(* IEC 61131-3 sources: AXOpen/src/showcase/app/SystemConstants (part 4) *)

TYPE
    kuka_rb1_DIO512_Output_Layout : STRUCT
        Signals_64_0 AT %X0.0 : BOOL;
        Signals_64_1 AT %X0.1 : BOOL;
        Signals_64_2 AT %X0.2 : BOOL;
        Signals_64_3 AT %X0.3 : BOOL;
        Signals_64_4 AT %X0.4 : BOOL;
        Signals_64_5 AT %X0.5 : BOOL;
        Signals_64_6 AT %X0.6 : BOOL;
        Signals_64_7 AT %X0.7 : BOOL;
        Signals_65_0 AT %X1.0 : BOOL;
        Signals_65_1 AT %X1.1 : BOOL;
        Signals_65_2 AT %X1.2 : BOOL;
        Signals_65_3 AT %X1.3 : BOOL;
        Signals_65_4 AT %X1.4 : BOOL;
        Signals_65_5 AT %X1.5 : BOOL;
        Signals_65_6 AT %X1.6 : BOOL;
        Signals_65_7 AT %X1.7 : BOOL;
        Signals_66_0 AT %X2.0 : BOOL;
        Signals_66_1 AT %X2.1 : BOOL;
        Signals_66_2 AT %X2.2 : BOOL;
        Signals_66_3 AT %X2.3 : BOOL;
        Signals_66_4 AT %X2.4 : BOOL;
        Signals_66_5 AT %X2.5 : BOOL;
        Signals_66_6 AT %X2.6 : BOOL;
        Signals_66_7 AT %X2.7 : BOOL;
        Signals_67_0 AT %X3.0 : BOOL;
        Signals_67_1 AT %X3.1 : BOOL;
        Signals_67_2 AT %X3.2 : BOOL;
        Signals_67_3 AT %X3.3 : BOOL;
        Signals_67_4 AT %X3.4 : BOOL;
        Signals_67_5 AT %X3.5 : BOOL;
        Signals_67_6 AT %X3.6 : BOOL;
        Signals_67_7 AT %X3.7 : BOOL;
        Signals_68_0 AT %X4.0 : BOOL;
        Signals_68_1 AT %X4.1 : BOOL;
        Signals_68_2 AT %X4.2 : BOOL;
        Signals_68_3 AT %X4.3 : BOOL;
        Signals_68_4 AT %X4.4 : BOOL;
        Signals_68_5 AT %X4.5 : BOOL;
        Signals_68_6 AT %X4.6 : BOOL;
        Signals_68_7 AT %X4.7 : BOOL;
        Signals_69_0 AT %X5.0 : BOOL;
        Signals_69_1 AT %X5.1 : BOOL;
        Signals_69_2 AT %X5.2 : BOOL;
        Signals_69_3 AT %X5.3 : BOOL;
        Signals_69_4 AT %X5.4 : BOOL;
        Signals_69_5 AT %X5.5 : BOOL;
        Signals_69_6 AT %X5.6 : BOOL;
        Signals_69_7 AT %X5.7 : BOOL;
        Signals_70_0 AT %X6.0 : BOOL;
        Signals_70_1 AT %X6.1 : BOOL;
        Signals_70_2 AT %X6.2 : BOOL;
        Signals_70_3 AT %X6.3 : BOOL;
        Signals_70_4 AT %X6.4 : BOOL;
        Signals_70_5 AT %X6.5 : BOOL;
        Signals_70_6 AT %X6.6 : BOOL;
        Signals_70_7 AT %X6.7 : BOOL;
        Signals_71_0 AT %X7.0 : BOOL;
        Signals_71_1 AT %X7.1 : BOOL;
        Signals_71_2 AT %X7.2 : BOOL;
        Signals_71_3 AT %X7.3 : BOOL;
        Signals_71_4 AT %X7.4 : BOOL;
        Signals_71_5 AT %X7.5 : BOOL;
        Signals_71_6 AT %X7.6 : BOOL;
        Signals_71_7 AT %X7.7 : BOOL;
        Signals_72_0 AT %X8.0 : BOOL;
        Signals_72_1 AT %X8.1 : BOOL;
        Signals_72_2 AT %X8.2 : BOOL;
        Signals_72_3 AT %X8.3 : BOOL;
        Signals_72_4 AT %X8.4 : BOOL;
        Signals_72_5 AT %X8.5 : BOOL;
        Signals_72_6 AT %X8.6 : BOOL;
        Signals_72_7 AT %X8.7 : BOOL;
        Signals_73_0 AT %X9.0 : BOOL;
        Signals_73_1 AT %X9.1 : BOOL;
        Signals_73_2 AT %X9.2 : BOOL;
        Signals_73_3 AT %X9.3 : BOOL;
        Signals_73_4 AT %X9.4 : BOOL;
        Signals_73_5 AT %X9.5 : BOOL;
        Signals_73_6 AT %X9.6 : BOOL;
        Signals_73_7 AT %X9.7 : BOOL;
        Signals_74_0 AT %X10.0 : BOOL;
        Signals_74_1 AT %X10.1 : BOOL;
        Signals_74_2 AT %X10.2 : BOOL;
        Signals_74_3 AT %X10.3 : BOOL;
        Signals_74_4 AT %X10.4 : BOOL;
        Signals_74_5 AT %X10.5 : BOOL;
        Signals_74_6 AT %X10.6 : BOOL;
        Signals_74_7 AT %X10.7 : BOOL;
        Signals_75_0 AT %X11.0 : BOOL;
        Signals_75_1 AT %X11.1 : BOOL;
        Signals_75_2 AT %X11.2 : BOOL;
        Signals_75_3 AT %X11.3 : BOOL;
        Signals_75_4 AT %X11.4 : BOOL;
        Signals_75_5 AT %X11.5 : BOOL;
        Signals_75_6 AT %X11.6 : BOOL;
        Signals_75_7 AT %X11.7 : BOOL;
        Signals_76_0 AT %X12.0 : BOOL;
        Signals_76_1 AT %X12.1 : BOOL;
        Signals_76_2 AT %X12.2 : BOOL;
        Signals_76_3 AT %X12.3 : BOOL;
        Signals_76_4 AT %X12.4 : BOOL;
        Signals_76_5 AT %X12.5 : BOOL;
        Signals_76_6 AT %X12.6 : BOOL;
        Signals_76_7 AT %X12.7 : BOOL;
        Signals_77_0 AT %X13.0 : BOOL;
        Signals_77_1 AT %X13.1 : BOOL;
        Signals_77_2 AT %X13.2 : BOOL;
        Signals_77_3 AT %X13.3 : BOOL;
        Signals_77_4 AT %X13.4 : BOOL;
        Signals_77_5 AT %X13.5 : BOOL;
        Signals_77_6 AT %X13.6 : BOOL;
        Signals_77_7 AT %X13.7 : BOOL;
        Signals_78_0 AT %X14.0 : BOOL;
        Signals_78_1 AT %X14.1 : BOOL;
        Signals_78_2 AT %X14.2 : BOOL;
        Signals_78_3 AT %X14.3 : BOOL;
        Signals_78_4 AT %X14.4 : BOOL;
        Signals_78_5 AT %X14.5 : BOOL;
        Signals_78_6 AT %X14.6 : BOOL;
        Signals_78_7 AT %X14.7 : BOOL;
        Signals_79_0 AT %X15.0 : BOOL;
        Signals_79_1 AT %X15.1 : BOOL;
        Signals_79_2 AT %X15.2 : BOOL;
        Signals_79_3 AT %X15.3 : BOOL;
        Signals_79_4 AT %X15.4 : BOOL;
        Signals_79_5 AT %X15.5 : BOOL;
        Signals_79_6 AT %X15.6 : BOOL;
        Signals_79_7 AT %X15.7 : BOOL;
        Signals_80_0 AT %X16.0 : BOOL;
        Signals_80_1 AT %X16.1 : BOOL;
        Signals_80_2 AT %X16.2 : BOOL;
        Signals_80_3 AT %X16.3 : BOOL;
        Signals_80_4 AT %X16.4 : BOOL;
        Signals_80_5 AT %X16.5 : BOOL;
        Signals_80_6 AT %X16.6 : BOOL;
        Signals_80_7 AT %X16.7 : BOOL;
        Signals_81_0 AT %X17.0 : BOOL;
        Signals_81_1 AT %X17.1 : BOOL;
        Signals_81_2 AT %X17.2 : BOOL;
        Signals_81_3 AT %X17.3 : BOOL;
        Signals_81_4 AT %X17.4 : BOOL;
        Signals_81_5 AT %X17.5 : BOOL;
        Signals_81_6 AT %X17.6 : BOOL;
        Signals_81_7 AT %X17.7 : BOOL;
        Signals_82_0 AT %X18.0 : BOOL;
        Signals_82_1 AT %X18.1 : BOOL;
        Signals_82_2 AT %X18.2 : BOOL;
        Signals_82_3 AT %X18.3 : BOOL;
        Signals_82_4 AT %X18.4 : BOOL;
        Signals_82_5 AT %X18.5 : BOOL;
        Signals_82_6 AT %X18.6 : BOOL;
        Signals_82_7 AT %X18.7 : BOOL;
        Signals_83_0 AT %X19.0 : BOOL;
        Signals_83_1 AT %X19.1 : BOOL;
        Signals_83_2 AT %X19.2 : BOOL;
        Signals_83_3 AT %X19.3 : BOOL;
        Signals_83_4 AT %X19.4 : BOOL;
        Signals_83_5 AT %X19.5 : BOOL;
        Signals_83_6 AT %X19.6 : BOOL;
        Signals_83_7 AT %X19.7 : BOOL;
        Signals_84_0 AT %X20.0 : BOOL;
        Signals_84_1 AT %X20.1 : BOOL;
        Signals_84_2 AT %X20.2 : BOOL;
        Signals_84_3 AT %X20.3 : BOOL;
        Signals_84_4 AT %X20.4 : BOOL;
        Signals_84_5 AT %X20.5 : BOOL;
        Signals_84_6 AT %X20.6 : BOOL;
        Signals_84_7 AT %X20.7 : BOOL;
        Signals_85_0 AT %X21.0 : BOOL;
        Signals_85_1 AT %X21.1 : BOOL;
        Signals_85_2 AT %X21.2 : BOOL;
        Signals_85_3 AT %X21.3 : BOOL;
        Signals_85_4 AT %X21.4 : BOOL;
        Signals_85_5 AT %X21.5 : BOOL;
        Signals_85_6 AT %X21.6 : BOOL;
        Signals_85_7 AT %X21.7 : BOOL;
        Signals_86_0 AT %X22.0 : BOOL;
        Signals_86_1 AT %X22.1 : BOOL;
        Signals_86_2 AT %X22.2 : BOOL;
        Signals_86_3 AT %X22.3 : BOOL;
        Signals_86_4 AT %X22.4 : BOOL;
        Signals_86_5 AT %X22.5 : BOOL;
        Signals_86_6 AT %X22.6 : BOOL;
        Signals_86_7 AT %X22.7 : BOOL;
        Signals_87_0 AT %X23.0 : BOOL;
        Signals_87_1 AT %X23.1 : BOOL;
        Signals_87_2 AT %X23.2 : BOOL;
        Signals_87_3 AT %X23.3 : BOOL;
        Signals_87_4 AT %X23.4 : BOOL;
        Signals_87_5 AT %X23.5 : BOOL;
        Signals_87_6 AT %X23.6 : BOOL;
        Signals_87_7 AT %X23.7 : BOOL;
        Signals_88_0 AT %X24.0 : BOOL;
        Signals_88_1 AT %X24.1 : BOOL;
        Signals_88_2 AT %X24.2 : BOOL;
        Signals_88_3 AT %X24.3 : BOOL;
        Signals_88_4 AT %X24.4 : BOOL;
        Signals_88_5 AT %X24.5 : BOOL;
        Signals_88_6 AT %X24.6 : BOOL;
        Signals_88_7 AT %X24.7 : BOOL;
        Signals_89_0 AT %X25.0 : BOOL;
        Signals_89_1 AT %X25.1 : BOOL;
        Signals_89_2 AT %X25.2 : BOOL;
        Signals_89_3 AT %X25.3 : BOOL;
        Signals_89_4 AT %X25.4 : BOOL;
        Signals_89_5 AT %X25.5 : BOOL;
        Signals_89_6 AT %X25.6 : BOOL;
        Signals_89_7 AT %X25.7 : BOOL;
        Signals_90_0 AT %X26.0 : BOOL;
        Signals_90_1 AT %X26.1 : BOOL;
        Signals_90_2 AT %X26.2 : BOOL;
        Signals_90_3 AT %X26.3 : BOOL;
        Signals_90_4 AT %X26.4 : BOOL;
        Signals_90_5 AT %X26.5 : BOOL;
        Signals_90_6 AT %X26.6 : BOOL;
        Signals_90_7 AT %X26.7 : BOOL;
        Signals_91_0 AT %X27.0 : BOOL;
        Signals_91_1 AT %X27.1 : BOOL;
        Signals_91_2 AT %X27.2 : BOOL;
        Signals_91_3 AT %X27.3 : BOOL;
        Signals_91_4 AT %X27.4 : BOOL;
        Signals_91_5 AT %X27.5 : BOOL;
        Signals_91_6 AT %X27.6 : BOOL;
        Signals_91_7 AT %X27.7 : BOOL;
        Signals_92_0 AT %X28.0 : BOOL;
        Signals_92_1 AT %X28.1 : BOOL;
        Signals_92_2 AT %X28.2 : BOOL;
        Signals_92_3 AT %X28.3 : BOOL;
        Signals_92_4 AT %X28.4 : BOOL;
        Signals_92_5 AT %X28.5 : BOOL;
        Signals_92_6 AT %X28.6 : BOOL;
        Signals_92_7 AT %X28.7 : BOOL;
        Signals_93_0 AT %X29.0 : BOOL;
        Signals_93_1 AT %X29.1 : BOOL;
        Signals_93_2 AT %X29.2 : BOOL;
        Signals_93_3 AT %X29.3 : BOOL;
        Signals_93_4 AT %X29.4 : BOOL;
        Signals_93_5 AT %X29.5 : BOOL;
        Signals_93_6 AT %X29.6 : BOOL;
        Signals_93_7 AT %X29.7 : BOOL;
        Signals_94_0 AT %X30.0 : BOOL;
        Signals_94_1 AT %X30.1 : BOOL;
        Signals_94_2 AT %X30.2 : BOOL;
        Signals_94_3 AT %X30.3 : BOOL;
        Signals_94_4 AT %X30.4 : BOOL;
        Signals_94_5 AT %X30.5 : BOOL;
        Signals_94_6 AT %X30.6 : BOOL;
        Signals_94_7 AT %X30.7 : BOOL;
        Signals_95_0 AT %X31.0 : BOOL;
        Signals_95_1 AT %X31.1 : BOOL;
        Signals_95_2 AT %X31.2 : BOOL;
        Signals_95_3 AT %X31.3 : BOOL;
        Signals_95_4 AT %X31.4 : BOOL;
        Signals_95_5 AT %X31.5 : BOOL;
        Signals_95_6 AT %X31.6 : BOOL;
        Signals_95_7 AT %X31.7 : BOOL;
        Signals_96_0 AT %X32.0 : BOOL;
        Signals_96_1 AT %X32.1 : BOOL;
        Signals_96_2 AT %X32.2 : BOOL;
        Signals_96_3 AT %X32.3 : BOOL;
        Signals_96_4 AT %X32.4 : BOOL;
        Signals_96_5 AT %X32.5 : BOOL;
        Signals_96_6 AT %X32.6 : BOOL;
        Signals_96_7 AT %X32.7 : BOOL;
        Signals_97_0 AT %X33.0 : BOOL;
        Signals_97_1 AT %X33.1 : BOOL;
        Signals_97_2 AT %X33.2 : BOOL;
        Signals_97_3 AT %X33.3 : BOOL;
        Signals_97_4 AT %X33.4 : BOOL;
        Signals_97_5 AT %X33.5 : BOOL;
        Signals_97_6 AT %X33.6 : BOOL;
        Signals_97_7 AT %X33.7 : BOOL;
        Signals_98_0 AT %X34.0 : BOOL;
        Signals_98_1 AT %X34.1 : BOOL;
        Signals_98_2 AT %X34.2 : BOOL;
        Signals_98_3 AT %X34.3 : BOOL;
        Signals_98_4 AT %X34.4 : BOOL;
        Signals_98_5 AT %X34.5 : BOOL;
        Signals_98_6 AT %X34.6 : BOOL;
        Signals_98_7 AT %X34.7 : BOOL;
        Signals_99_0 AT %X35.0 : BOOL;
        Signals_99_1 AT %X35.1 : BOOL;
        Signals_99_2 AT %X35.2 : BOOL;
        Signals_99_3 AT %X35.3 : BOOL;
        Signals_99_4 AT %X35.4 : BOOL;
        Signals_99_5 AT %X35.5 : BOOL;
        Signals_99_6 AT %X35.6 : BOOL;
        Signals_99_7 AT %X35.7 : BOOL;
        Signals_100_0 AT %X36.0 : BOOL;
        Signals_100_1 AT %X36.1 : BOOL;
        Signals_100_2 AT %X36.2 : BOOL;
        Signals_100_3 AT %X36.3 : BOOL;
        Signals_100_4 AT %X36.4 : BOOL;
        Signals_100_5 AT %X36.5 : BOOL;
        Signals_100_6 AT %X36.6 : BOOL;
        Signals_100_7 AT %X36.7 : BOOL;
        Signals_101_0 AT %X37.0 : BOOL;
        Signals_101_1 AT %X37.1 : BOOL;
        Signals_101_2 AT %X37.2 : BOOL;
        Signals_101_3 AT %X37.3 : BOOL;
        Signals_101_4 AT %X37.4 : BOOL;
        Signals_101_5 AT %X37.5 : BOOL;
        Signals_101_6 AT %X37.6 : BOOL;
        Signals_101_7 AT %X37.7 : BOOL;
        Signals_102_0 AT %X38.0 : BOOL;
        Signals_102_1 AT %X38.1 : BOOL;
        Signals_102_2 AT %X38.2 : BOOL;
        Signals_102_3 AT %X38.3 : BOOL;
        Signals_102_4 AT %X38.4 : BOOL;
        Signals_102_5 AT %X38.5 : BOOL;
        Signals_102_6 AT %X38.6 : BOOL;
        Signals_102_7 AT %X38.7 : BOOL;
        Signals_103_0 AT %X39.0 : BOOL;
        Signals_103_1 AT %X39.1 : BOOL;
        Signals_103_2 AT %X39.2 : BOOL;
        Signals_103_3 AT %X39.3 : BOOL;
        Signals_103_4 AT %X39.4 : BOOL;
        Signals_103_5 AT %X39.5 : BOOL;
        Signals_103_6 AT %X39.6 : BOOL;
        Signals_103_7 AT %X39.7 : BOOL;
        Signals_104_0 AT %X40.0 : BOOL;
        Signals_104_1 AT %X40.1 : BOOL;
        Signals_104_2 AT %X40.2 : BOOL;
        Signals_104_3 AT %X40.3 : BOOL;
        Signals_104_4 AT %X40.4 : BOOL;
        Signals_104_5 AT %X40.5 : BOOL;
        Signals_104_6 AT %X40.6 : BOOL;
        Signals_104_7 AT %X40.7 : BOOL;
        Signals_105_0 AT %X41.0 : BOOL;
        Signals_105_1 AT %X41.1 : BOOL;
        Signals_105_2 AT %X41.2 : BOOL;
        Signals_105_3 AT %X41.3 : BOOL;
        Signals_105_4 AT %X41.4 : BOOL;
        Signals_105_5 AT %X41.5 : BOOL;
        Signals_105_6 AT %X41.6 : BOOL;
        Signals_105_7 AT %X41.7 : BOOL;
        Signals_106_0 AT %X42.0 : BOOL;
        Signals_106_1 AT %X42.1 : BOOL;
        Signals_106_2 AT %X42.2 : BOOL;
        Signals_106_3 AT %X42.3 : BOOL;
        Signals_106_4 AT %X42.4 : BOOL;
        Signals_106_5 AT %X42.5 : BOOL;
        Signals_106_6 AT %X42.6 : BOOL;
        Signals_106_7 AT %X42.7 : BOOL;
        Signals_107_0 AT %X43.0 : BOOL;
        Signals_107_1 AT %X43.1 : BOOL;
        Signals_107_2 AT %X43.2 : BOOL;
        Signals_107_3 AT %X43.3 : BOOL;
        Signals_107_4 AT %X43.4 : BOOL;
        Signals_107_5 AT %X43.5 : BOOL;
        Signals_107_6 AT %X43.6 : BOOL;
        Signals_107_7 AT %X43.7 : BOOL;
        Signals_108_0 AT %X44.0 : BOOL;
        Signals_108_1 AT %X44.1 : BOOL;
        Signals_108_2 AT %X44.2 : BOOL;
        Signals_108_3 AT %X44.3 : BOOL;
        Signals_108_4 AT %X44.4 : BOOL;
        Signals_108_5 AT %X44.5 : BOOL;
        Signals_108_6 AT %X44.6 : BOOL;
        Signals_108_7 AT %X44.7 : BOOL;
        Signals_109_0 AT %X45.0 : BOOL;
        Signals_109_1 AT %X45.1 : BOOL;
        Signals_109_2 AT %X45.2 : BOOL;
        Signals_109_3 AT %X45.3 : BOOL;
        Signals_109_4 AT %X45.4 : BOOL;
        Signals_109_5 AT %X45.5 : BOOL;
        Signals_109_6 AT %X45.6 : BOOL;
        Signals_109_7 AT %X45.7 : BOOL;
        Signals_110_0 AT %X46.0 : BOOL;
        Signals_110_1 AT %X46.1 : BOOL;
        Signals_110_2 AT %X46.2 : BOOL;
        Signals_110_3 AT %X46.3 : BOOL;
        Signals_110_4 AT %X46.4 : BOOL;
        Signals_110_5 AT %X46.5 : BOOL;
        Signals_110_6 AT %X46.6 : BOOL;
        Signals_110_7 AT %X46.7 : BOOL;
        Signals_111_0 AT %X47.0 : BOOL;
        Signals_111_1 AT %X47.1 : BOOL;
        Signals_111_2 AT %X47.2 : BOOL;
        Signals_111_3 AT %X47.3 : BOOL;
        Signals_111_4 AT %X47.4 : BOOL;
        Signals_111_5 AT %X47.5 : BOOL;
        Signals_111_6 AT %X47.6 : BOOL;
        Signals_111_7 AT %X47.7 : BOOL;
        Signals_112_0 AT %X48.0 : BOOL;
        Signals_112_1 AT %X48.1 : BOOL;
        Signals_112_2 AT %X48.2 : BOOL;
        Signals_112_3 AT %X48.3 : BOOL;
        Signals_112_4 AT %X48.4 : BOOL;
        Signals_112_5 AT %X48.5 : BOOL;
        Signals_112_6 AT %X48.6 : BOOL;
        Signals_112_7 AT %X48.7 : BOOL;
        Signals_113_0 AT %X49.0 : BOOL;
        Signals_113_1 AT %X49.1 : BOOL;
        Signals_113_2 AT %X49.2 : BOOL;
        Signals_113_3 AT %X49.3 : BOOL;
        Signals_113_4 AT %X49.4 : BOOL;
        Signals_113_5 AT %X49.5 : BOOL;
        Signals_113_6 AT %X49.6 : BOOL;
        Signals_113_7 AT %X49.7 : BOOL;
        Signals_114_0 AT %X50.0 : BOOL;
        Signals_114_1 AT %X50.1 : BOOL;
        Signals_114_2 AT %X50.2 : BOOL;
        Signals_114_3 AT %X50.3 : BOOL;
        Signals_114_4 AT %X50.4 : BOOL;
        Signals_114_5 AT %X50.5 : BOOL;
        Signals_114_6 AT %X50.6 : BOOL;
        Signals_114_7 AT %X50.7 : BOOL;
        Signals_115_0 AT %X51.0 : BOOL;
        Signals_115_1 AT %X51.1 : BOOL;
        Signals_115_2 AT %X51.2 : BOOL;
        Signals_115_3 AT %X51.3 : BOOL;
        Signals_115_4 AT %X51.4 : BOOL;
        Signals_115_5 AT %X51.5 : BOOL;
        Signals_115_6 AT %X51.6 : BOOL;
        Signals_115_7 AT %X51.7 : BOOL;
        Signals_116_0 AT %X52.0 : BOOL;
        Signals_116_1 AT %X52.1 : BOOL;
        Signals_116_2 AT %X52.2 : BOOL;
        Signals_116_3 AT %X52.3 : BOOL;
        Signals_116_4 AT %X52.4 : BOOL;
        Signals_116_5 AT %X52.5 : BOOL;
        Signals_116_6 AT %X52.6 : BOOL;
        Signals_116_7 AT %X52.7 : BOOL;
        Signals_117_0 AT %X53.0 : BOOL;
        Signals_117_1 AT %X53.1 : BOOL;
        Signals_117_2 AT %X53.2 : BOOL;
        Signals_117_3 AT %X53.3 : BOOL;
        Signals_117_4 AT %X53.4 : BOOL;
        Signals_117_5 AT %X53.5 : BOOL;
        Signals_117_6 AT %X53.6 : BOOL;
        Signals_117_7 AT %X53.7 : BOOL;
        Signals_118_0 AT %X54.0 : BOOL;
        Signals_118_1 AT %X54.1 : BOOL;
        Signals_118_2 AT %X54.2 : BOOL;
        Signals_118_3 AT %X54.3 : BOOL;
        Signals_118_4 AT %X54.4 : BOOL;
        Signals_118_5 AT %X54.5 : BOOL;
        Signals_118_6 AT %X54.6 : BOOL;
        Signals_118_7 AT %X54.7 : BOOL;
        Signals_119_0 AT %X55.0 : BOOL;
        Signals_119_1 AT %X55.1 : BOOL;
        Signals_119_2 AT %X55.2 : BOOL;
        Signals_119_3 AT %X55.3 : BOOL;
        Signals_119_4 AT %X55.4 : BOOL;
        Signals_119_5 AT %X55.5 : BOOL;
        Signals_119_6 AT %X55.6 : BOOL;
        Signals_119_7 AT %X55.7 : BOOL;
        Signals_120_0 AT %X56.0 : BOOL;
        Signals_120_1 AT %X56.1 : BOOL;
        Signals_120_2 AT %X56.2 : BOOL;
        Signals_120_3 AT %X56.3 : BOOL;
        Signals_120_4 AT %X56.4 : BOOL;
        Signals_120_5 AT %X56.5 : BOOL;
        Signals_120_6 AT %X56.6 : BOOL;
        Signals_120_7 AT %X56.7 : BOOL;
        Signals_121_0 AT %X57.0 : BOOL;
        Signals_121_1 AT %X57.1 : BOOL;
        Signals_121_2 AT %X57.2 : BOOL;
        Signals_121_3 AT %X57.3 : BOOL;
        Signals_121_4 AT %X57.4 : BOOL;
        Signals_121_5 AT %X57.5 : BOOL;
        Signals_121_6 AT %X57.6 : BOOL;
        Signals_121_7 AT %X57.7 : BOOL;
        Signals_122_0 AT %X58.0 : BOOL;
        Signals_122_1 AT %X58.1 : BOOL;
        Signals_122_2 AT %X58.2 : BOOL;
        Signals_122_3 AT %X58.3 : BOOL;
        Signals_122_4 AT %X58.4 : BOOL;
        Signals_122_5 AT %X58.5 : BOOL;
        Signals_122_6 AT %X58.6 : BOOL;
        Signals_122_7 AT %X58.7 : BOOL;
        Signals_123_0 AT %X59.0 : BOOL;
        Signals_123_1 AT %X59.1 : BOOL;
        Signals_123_2 AT %X59.2 : BOOL;
        Signals_123_3 AT %X59.3 : BOOL;
        Signals_123_4 AT %X59.4 : BOOL;
        Signals_123_5 AT %X59.5 : BOOL;
        Signals_123_6 AT %X59.6 : BOOL;
        Signals_123_7 AT %X59.7 : BOOL;
        Signals_124_0 AT %X60.0 : BOOL;
        Signals_124_1 AT %X60.1 : BOOL;
        Signals_124_2 AT %X60.2 : BOOL;
        Signals_124_3 AT %X60.3 : BOOL;
        Signals_124_4 AT %X60.4 : BOOL;
        Signals_124_5 AT %X60.5 : BOOL;
        Signals_124_6 AT %X60.6 : BOOL;
        Signals_124_7 AT %X60.7 : BOOL;
        Signals_125_0 AT %X61.0 : BOOL;
        Signals_125_1 AT %X61.1 : BOOL;
        Signals_125_2 AT %X61.2 : BOOL;
        Signals_125_3 AT %X61.3 : BOOL;
        Signals_125_4 AT %X61.4 : BOOL;
        Signals_125_5 AT %X61.5 : BOOL;
        Signals_125_6 AT %X61.6 : BOOL;
        Signals_125_7 AT %X61.7 : BOOL;
        Signals_126_0 AT %X62.0 : BOOL;
        Signals_126_1 AT %X62.1 : BOOL;
        Signals_126_2 AT %X62.2 : BOOL;
        Signals_126_3 AT %X62.3 : BOOL;
        Signals_126_4 AT %X62.4 : BOOL;
        Signals_126_5 AT %X62.5 : BOOL;
        Signals_126_6 AT %X62.6 : BOOL;
        Signals_126_7 AT %X62.7 : BOOL;
        Signals_127_0 AT %X63.0 : BOOL;
        Signals_127_1 AT %X63.1 : BOOL;
        Signals_127_2 AT %X63.2 : BOOL;
        Signals_127_3 AT %X63.3 : BOOL;
        Signals_127_4 AT %X63.4 : BOOL;
        Signals_127_5 AT %X63.5 : BOOL;
        Signals_127_6 AT %X63.6 : BOOL;
        Signals_127_7 AT %X63.7 : BOOL;
    END_STRUCT;
END_TYPE

TYPE
    kuka_rb2_DIO512_Input_Layout : STRUCT
        Signals_0_0 AT %X0.0 : BOOL;
        Signals_0_1 AT %X0.1 : BOOL;
        Signals_0_2 AT %X0.2 : BOOL;
        Signals_0_3 AT %X0.3 : BOOL;
        Signals_0_4 AT %X0.4 : BOOL;
        Signals_0_5 AT %X0.5 : BOOL;
        Signals_0_6 AT %X0.6 : BOOL;
        Signals_0_7 AT %X0.7 : BOOL;
        Signals_1_0 AT %X1.0 : BOOL;
        Signals_1_1 AT %X1.1 : BOOL;
        Signals_1_2 AT %X1.2 : BOOL;
        Signals_1_3 AT %X1.3 : BOOL;
        Signals_1_4 AT %X1.4 : BOOL;
        Signals_1_5 AT %X1.5 : BOOL;
        Signals_1_6 AT %X1.6 : BOOL;
        Signals_1_7 AT %X1.7 : BOOL;
        Signals_2_0 AT %X2.0 : BOOL;
        Signals_2_1 AT %X2.1 : BOOL;
        Signals_2_2 AT %X2.2 : BOOL;
        Signals_2_3 AT %X2.3 : BOOL;
        Signals_2_4 AT %X2.4 : BOOL;
        Signals_2_5 AT %X2.5 : BOOL;
        Signals_2_6 AT %X2.6 : BOOL;
        Signals_2_7 AT %X2.7 : BOOL;
        Signals_3_0 AT %X3.0 : BOOL;
        Signals_3_1 AT %X3.1 : BOOL;
        Signals_3_2 AT %X3.2 : BOOL;
        Signals_3_3 AT %X3.3 : BOOL;
        Signals_3_4 AT %X3.4 : BOOL;
        Signals_3_5 AT %X3.5 : BOOL;
        Signals_3_6 AT %X3.6 : BOOL;
        Signals_3_7 AT %X3.7 : BOOL;
        Signals_4_0 AT %X4.0 : BOOL;
        Signals_4_1 AT %X4.1 : BOOL;
        Signals_4_2 AT %X4.2 : BOOL;
        Signals_4_3 AT %X4.3 : BOOL;
        Signals_4_4 AT %X4.4 : BOOL;
        Signals_4_5 AT %X4.5 : BOOL;
        Signals_4_6 AT %X4.6 : BOOL;
        Signals_4_7 AT %X4.7 : BOOL;
        Signals_5_0 AT %X5.0 : BOOL;
        Signals_5_1 AT %X5.1 : BOOL;
        Signals_5_2 AT %X5.2 : BOOL;
        Signals_5_3 AT %X5.3 : BOOL;
        Signals_5_4 AT %X5.4 : BOOL;
        Signals_5_5 AT %X5.5 : BOOL;
        Signals_5_6 AT %X5.6 : BOOL;
        Signals_5_7 AT %X5.7 : BOOL;
        Signals_6_0 AT %X6.0 : BOOL;
        Signals_6_1 AT %X6.1 : BOOL;
        Signals_6_2 AT %X6.2 : BOOL;
        Signals_6_3 AT %X6.3 : BOOL;
        Signals_6_4 AT %X6.4 : BOOL;
        Signals_6_5 AT %X6.5 : BOOL;
        Signals_6_6 AT %X6.6 : BOOL;
        Signals_6_7 AT %X6.7 : BOOL;
        Signals_7_0 AT %X7.0 : BOOL;
        Signals_7_1 AT %X7.1 : BOOL;
        Signals_7_2 AT %X7.2 : BOOL;
        Signals_7_3 AT %X7.3 : BOOL;
        Signals_7_4 AT %X7.4 : BOOL;
        Signals_7_5 AT %X7.5 : BOOL;
        Signals_7_6 AT %X7.6 : BOOL;
        Signals_7_7 AT %X7.7 : BOOL;
        Signals_8_0 AT %X8.0 : BOOL;
        Signals_8_1 AT %X8.1 : BOOL;
        Signals_8_2 AT %X8.2 : BOOL;
        Signals_8_3 AT %X8.3 : BOOL;
        Signals_8_4 AT %X8.4 : BOOL;
        Signals_8_5 AT %X8.5 : BOOL;
        Signals_8_6 AT %X8.6 : BOOL;
        Signals_8_7 AT %X8.7 : BOOL;
        Signals_9_0 AT %X9.0 : BOOL;
        Signals_9_1 AT %X9.1 : BOOL;
        Signals_9_2 AT %X9.2 : BOOL;
        Signals_9_3 AT %X9.3 : BOOL;
        Signals_9_4 AT %X9.4 : BOOL;
        Signals_9_5 AT %X9.5 : BOOL;
        Signals_9_6 AT %X9.6 : BOOL;
        Signals_9_7 AT %X9.7 : BOOL;
        Signals_10_0 AT %X10.0 : BOOL;
        Signals_10_1 AT %X10.1 : BOOL;
        Signals_10_2 AT %X10.2 : BOOL;
        Signals_10_3 AT %X10.3 : BOOL;
        Signals_10_4 AT %X10.4 : BOOL;
        Signals_10_5 AT %X10.5 : BOOL;
        Signals_10_6 AT %X10.6 : BOOL;
        Signals_10_7 AT %X10.7 : BOOL;
        Signals_11_0 AT %X11.0 : BOOL;
        Signals_11_1 AT %X11.1 : BOOL;
        Signals_11_2 AT %X11.2 : BOOL;
        Signals_11_3 AT %X11.3 : BOOL;
        Signals_11_4 AT %X11.4 : BOOL;
        Signals_11_5 AT %X11.5 : BOOL;
        Signals_11_6 AT %X11.6 : BOOL;
        Signals_11_7 AT %X11.7 : BOOL;
        Signals_12_0 AT %X12.0 : BOOL;
        Signals_12_1 AT %X12.1 : BOOL;
        Signals_12_2 AT %X12.2 : BOOL;
        Signals_12_3 AT %X12.3 : BOOL;
        Signals_12_4 AT %X12.4 : BOOL;
        Signals_12_5 AT %X12.5 : BOOL;
        Signals_12_6 AT %X12.6 : BOOL;
        Signals_12_7 AT %X12.7 : BOOL;
        Signals_13_0 AT %X13.0 : BOOL;
        Signals_13_1 AT %X13.1 : BOOL;
        Signals_13_2 AT %X13.2 : BOOL;
        Signals_13_3 AT %X13.3 : BOOL;
        Signals_13_4 AT %X13.4 : BOOL;
        Signals_13_5 AT %X13.5 : BOOL;
        Signals_13_6 AT %X13.6 : BOOL;
        Signals_13_7 AT %X13.7 : BOOL;
        Signals_14_0 AT %X14.0 : BOOL;
        Signals_14_1 AT %X14.1 : BOOL;
        Signals_14_2 AT %X14.2 : BOOL;
        Signals_14_3 AT %X14.3 : BOOL;
        Signals_14_4 AT %X14.4 : BOOL;
        Signals_14_5 AT %X14.5 : BOOL;
        Signals_14_6 AT %X14.6 : BOOL;
        Signals_14_7 AT %X14.7 : BOOL;
        Signals_15_0 AT %X15.0 : BOOL;
        Signals_15_1 AT %X15.1 : BOOL;
        Signals_15_2 AT %X15.2 : BOOL;
        Signals_15_3 AT %X15.3 : BOOL;
        Signals_15_4 AT %X15.4 : BOOL;
        Signals_15_5 AT %X15.5 : BOOL;
        Signals_15_6 AT %X15.6 : BOOL;
        Signals_15_7 AT %X15.7 : BOOL;
        Signals_16_0 AT %X16.0 : BOOL;
        Signals_16_1 AT %X16.1 : BOOL;
        Signals_16_2 AT %X16.2 : BOOL;
        Signals_16_3 AT %X16.3 : BOOL;
        Signals_16_4 AT %X16.4 : BOOL;
        Signals_16_5 AT %X16.5 : BOOL;
        Signals_16_6 AT %X16.6 : BOOL;
        Signals_16_7 AT %X16.7 : BOOL;
        Signals_17_0 AT %X17.0 : BOOL;
        Signals_17_1 AT %X17.1 : BOOL;
        Signals_17_2 AT %X17.2 : BOOL;
        Signals_17_3 AT %X17.3 : BOOL;
        Signals_17_4 AT %X17.4 : BOOL;
        Signals_17_5 AT %X17.5 : BOOL;
        Signals_17_6 AT %X17.6 : BOOL;
        Signals_17_7 AT %X17.7 : BOOL;
        Signals_18_0 AT %X18.0 : BOOL;
        Signals_18_1 AT %X18.1 : BOOL;
        Signals_18_2 AT %X18.2 : BOOL;
        Signals_18_3 AT %X18.3 : BOOL;
        Signals_18_4 AT %X18.4 : BOOL;
        Signals_18_5 AT %X18.5 : BOOL;
        Signals_18_6 AT %X18.6 : BOOL;
        Signals_18_7 AT %X18.7 : BOOL;
        Signals_19_0 AT %X19.0 : BOOL;
        Signals_19_1 AT %X19.1 : BOOL;
        Signals_19_2 AT %X19.2 : BOOL;
        Signals_19_3 AT %X19.3 : BOOL;
        Signals_19_4 AT %X19.4 : BOOL;
        Signals_19_5 AT %X19.5 : BOOL;
        Signals_19_6 AT %X19.6 : BOOL;
        Signals_19_7 AT %X19.7 : BOOL;
        Signals_20_0 AT %X20.0 : BOOL;
        Signals_20_1 AT %X20.1 : BOOL;
        Signals_20_2 AT %X20.2 : BOOL;
        Signals_20_3 AT %X20.3 : BOOL;
        Signals_20_4 AT %X20.4 : BOOL;
        Signals_20_5 AT %X20.5 : BOOL;
        Signals_20_6 AT %X20.6 : BOOL;
        Signals_20_7 AT %X20.7 : BOOL;
        Signals_21_0 AT %X21.0 : BOOL;
        Signals_21_1 AT %X21.1 : BOOL;
        Signals_21_2 AT %X21.2 : BOOL;
        Signals_21_3 AT %X21.3 : BOOL;
        Signals_21_4 AT %X21.4 : BOOL;
        Signals_21_5 AT %X21.5 : BOOL;
        Signals_21_6 AT %X21.6 : BOOL;
        Signals_21_7 AT %X21.7 : BOOL;
        Signals_22_0 AT %X22.0 : BOOL;
        Signals_22_1 AT %X22.1 : BOOL;
        Signals_22_2 AT %X22.2 : BOOL;
        Signals_22_3 AT %X22.3 : BOOL;
        Signals_22_4 AT %X22.4 : BOOL;
        Signals_22_5 AT %X22.5 : BOOL;
        Signals_22_6 AT %X22.6 : BOOL;
        Signals_22_7 AT %X22.7 : BOOL;
        Signals_23_0 AT %X23.0 : BOOL;
        Signals_23_1 AT %X23.1 : BOOL;
        Signals_23_2 AT %X23.2 : BOOL;
        Signals_23_3 AT %X23.3 : BOOL;
        Signals_23_4 AT %X23.4 : BOOL;
        Signals_23_5 AT %X23.5 : BOOL;
        Signals_23_6 AT %X23.6 : BOOL;
        Signals_23_7 AT %X23.7 : BOOL;
        Signals_24_0 AT %X24.0 : BOOL;
        Signals_24_1 AT %X24.1 : BOOL;
        Signals_24_2 AT %X24.2 : BOOL;
        Signals_24_3 AT %X24.3 : BOOL;
        Signals_24_4 AT %X24.4 : BOOL;
        Signals_24_5 AT %X24.5 : BOOL;
        Signals_24_6 AT %X24.6 : BOOL;
        Signals_24_7 AT %X24.7 : BOOL;
        Signals_25_0 AT %X25.0 : BOOL;
        Signals_25_1 AT %X25.1 : BOOL;
        Signals_25_2 AT %X25.2 : BOOL;
        Signals_25_3 AT %X25.3 : BOOL;
        Signals_25_4 AT %X25.4 : BOOL;
        Signals_25_5 AT %X25.5 : BOOL;
        Signals_25_6 AT %X25.6 : BOOL;
        Signals_25_7 AT %X25.7 : BOOL;
        Signals_26_0 AT %X26.0 : BOOL;
        Signals_26_1 AT %X26.1 : BOOL;
        Signals_26_2 AT %X26.2 : BOOL;
        Signals_26_3 AT %X26.3 : BOOL;
        Signals_26_4 AT %X26.4 : BOOL;
        Signals_26_5 AT %X26.5 : BOOL;
        Signals_26_6 AT %X26.6 : BOOL;
        Signals_26_7 AT %X26.7 : BOOL;
        Signals_27_0 AT %X27.0 : BOOL;
        Signals_27_1 AT %X27.1 : BOOL;
        Signals_27_2 AT %X27.2 : BOOL;
        Signals_27_3 AT %X27.3 : BOOL;
        Signals_27_4 AT %X27.4 : BOOL;
        Signals_27_5 AT %X27.5 : BOOL;
        Signals_27_6 AT %X27.6 : BOOL;
        Signals_27_7 AT %X27.7 : BOOL;
        Signals_28_0 AT %X28.0 : BOOL;
        Signals_28_1 AT %X28.1 : BOOL;
        Signals_28_2 AT %X28.2 : BOOL;
        Signals_28_3 AT %X28.3 : BOOL;
        Signals_28_4 AT %X28.4 : BOOL;
        Signals_28_5 AT %X28.5 : BOOL;
        Signals_28_6 AT %X28.6 : BOOL;
        Signals_28_7 AT %X28.7 : BOOL;
        Signals_29_0 AT %X29.0 : BOOL;
        Signals_29_1 AT %X29.1 : BOOL;
        Signals_29_2 AT %X29.2 : BOOL;
        Signals_29_3 AT %X29.3 : BOOL;
        Signals_29_4 AT %X29.4 : BOOL;
        Signals_29_5 AT %X29.5 : BOOL;
        Signals_29_6 AT %X29.6 : BOOL;
        Signals_29_7 AT %X29.7 : BOOL;
        Signals_30_0 AT %X30.0 : BOOL;
        Signals_30_1 AT %X30.1 : BOOL;
        Signals_30_2 AT %X30.2 : BOOL;
        Signals_30_3 AT %X30.3 : BOOL;
        Signals_30_4 AT %X30.4 : BOOL;
        Signals_30_5 AT %X30.5 : BOOL;
        Signals_30_6 AT %X30.6 : BOOL;
        Signals_30_7 AT %X30.7 : BOOL;
        Signals_31_0 AT %X31.0 : BOOL;
        Signals_31_1 AT %X31.1 : BOOL;
        Signals_31_2 AT %X31.2 : BOOL;
        Signals_31_3 AT %X31.3 : BOOL;
        Signals_31_4 AT %X31.4 : BOOL;
        Signals_31_5 AT %X31.5 : BOOL;
        Signals_31_6 AT %X31.6 : BOOL;
        Signals_31_7 AT %X31.7 : BOOL;
        Signals_32_0 AT %X32.0 : BOOL;
        Signals_32_1 AT %X32.1 : BOOL;
        Signals_32_2 AT %X32.2 : BOOL;
        Signals_32_3 AT %X32.3 : BOOL;
        Signals_32_4 AT %X32.4 : BOOL;
        Signals_32_5 AT %X32.5 : BOOL;
        Signals_32_6 AT %X32.6 : BOOL;
        Signals_32_7 AT %X32.7 : BOOL;
        Signals_33_0 AT %X33.0 : BOOL;
        Signals_33_1 AT %X33.1 : BOOL;
        Signals_33_2 AT %X33.2 : BOOL;
        Signals_33_3 AT %X33.3 : BOOL;
        Signals_33_4 AT %X33.4 : BOOL;
        Signals_33_5 AT %X33.5 : BOOL;
        Signals_33_6 AT %X33.6 : BOOL;
        Signals_33_7 AT %X33.7 : BOOL;
        Signals_34_0 AT %X34.0 : BOOL;
        Signals_34_1 AT %X34.1 : BOOL;
        Signals_34_2 AT %X34.2 : BOOL;
        Signals_34_3 AT %X34.3 : BOOL;
        Signals_34_4 AT %X34.4 : BOOL;
        Signals_34_5 AT %X34.5 : BOOL;
        Signals_34_6 AT %X34.6 : BOOL;
        Signals_34_7 AT %X34.7 : BOOL;
        Signals_35_0 AT %X35.0 : BOOL;
        Signals_35_1 AT %X35.1 : BOOL;
        Signals_35_2 AT %X35.2 : BOOL;
        Signals_35_3 AT %X35.3 : BOOL;
        Signals_35_4 AT %X35.4 : BOOL;
        Signals_35_5 AT %X35.5 : BOOL;
        Signals_35_6 AT %X35.6 : BOOL;
        Signals_35_7 AT %X35.7 : BOOL;
        Signals_36_0 AT %X36.0 : BOOL;
        Signals_36_1 AT %X36.1 : BOOL;
        Signals_36_2 AT %X36.2 : BOOL;
        Signals_36_3 AT %X36.3 : BOOL;
        Signals_36_4 AT %X36.4 : BOOL;
        Signals_36_5 AT %X36.5 : BOOL;
        Signals_36_6 AT %X36.6 : BOOL;
        Signals_36_7 AT %X36.7 : BOOL;
        Signals_37_0 AT %X37.0 : BOOL;
        Signals_37_1 AT %X37.1 : BOOL;
        Signals_37_2 AT %X37.2 : BOOL;
        Signals_37_3 AT %X37.3 : BOOL;
        Signals_37_4 AT %X37.4 : BOOL;
        Signals_37_5 AT %X37.5 : BOOL;
        Signals_37_6 AT %X37.6 : BOOL;
        Signals_37_7 AT %X37.7 : BOOL;
        Signals_38_0 AT %X38.0 : BOOL;
        Signals_38_1 AT %X38.1 : BOOL;
        Signals_38_2 AT %X38.2 : BOOL;
        Signals_38_3 AT %X38.3 : BOOL;
        Signals_38_4 AT %X38.4 : BOOL;
        Signals_38_5 AT %X38.5 : BOOL;
        Signals_38_6 AT %X38.6 : BOOL;
        Signals_38_7 AT %X38.7 : BOOL;
        Signals_39_0 AT %X39.0 : BOOL;
        Signals_39_1 AT %X39.1 : BOOL;
        Signals_39_2 AT %X39.2 : BOOL;
        Signals_39_3 AT %X39.3 : BOOL;
        Signals_39_4 AT %X39.4 : BOOL;
        Signals_39_5 AT %X39.5 : BOOL;
        Signals_39_6 AT %X39.6 : BOOL;
        Signals_39_7 AT %X39.7 : BOOL;
        Signals_40_0 AT %X40.0 : BOOL;
        Signals_40_1 AT %X40.1 : BOOL;
        Signals_40_2 AT %X40.2 : BOOL;
        Signals_40_3 AT %X40.3 : BOOL;
        Signals_40_4 AT %X40.4 : BOOL;
        Signals_40_5 AT %X40.5 : BOOL;
        Signals_40_6 AT %X40.6 : BOOL;
        Signals_40_7 AT %X40.7 : BOOL;
        Signals_41_0 AT %X41.0 : BOOL;
        Signals_41_1 AT %X41.1 : BOOL;
        Signals_41_2 AT %X41.2 : BOOL;
        Signals_41_3 AT %X41.3 : BOOL;
        Signals_41_4 AT %X41.4 : BOOL;
        Signals_41_5 AT %X41.5 : BOOL;
        Signals_41_6 AT %X41.6 : BOOL;
        Signals_41_7 AT %X41.7 : BOOL;
        Signals_42_0 AT %X42.0 : BOOL;
        Signals_42_1 AT %X42.1 : BOOL;
        Signals_42_2 AT %X42.2 : BOOL;
        Signals_42_3 AT %X42.3 : BOOL;
        Signals_42_4 AT %X42.4 : BOOL;
        Signals_42_5 AT %X42.5 : BOOL;
        Signals_42_6 AT %X42.6 : BOOL;
        Signals_42_7 AT %X42.7 : BOOL;
        Signals_43_0 AT %X43.0 : BOOL;
        Signals_43_1 AT %X43.1 : BOOL;
        Signals_43_2 AT %X43.2 : BOOL;
        Signals_43_3 AT %X43.3 : BOOL;
        Signals_43_4 AT %X43.4 : BOOL;
        Signals_43_5 AT %X43.5 : BOOL;
        Signals_43_6 AT %X43.6 : BOOL;
        Signals_43_7 AT %X43.7 : BOOL;
        Signals_44_0 AT %X44.0 : BOOL;
        Signals_44_1 AT %X44.1 : BOOL;
        Signals_44_2 AT %X44.2 : BOOL;
        Signals_44_3 AT %X44.3 : BOOL;
        Signals_44_4 AT %X44.4 : BOOL;
        Signals_44_5 AT %X44.5 : BOOL;
        Signals_44_6 AT %X44.6 : BOOL;
        Signals_44_7 AT %X44.7 : BOOL;
        Signals_45_0 AT %X45.0 : BOOL;
        Signals_45_1 AT %X45.1 : BOOL;
        Signals_45_2 AT %X45.2 : BOOL;
        Signals_45_3 AT %X45.3 : BOOL;
        Signals_45_4 AT %X45.4 : BOOL;
        Signals_45_5 AT %X45.5 : BOOL;
        Signals_45_6 AT %X45.6 : BOOL;
        Signals_45_7 AT %X45.7 : BOOL;
        Signals_46_0 AT %X46.0 : BOOL;
        Signals_46_1 AT %X46.1 : BOOL;
        Signals_46_2 AT %X46.2 : BOOL;
        Signals_46_3 AT %X46.3 : BOOL;
        Signals_46_4 AT %X46.4 : BOOL;
        Signals_46_5 AT %X46.5 : BOOL;
        Signals_46_6 AT %X46.6 : BOOL;
        Signals_46_7 AT %X46.7 : BOOL;
        Signals_47_0 AT %X47.0 : BOOL;
        Signals_47_1 AT %X47.1 : BOOL;
        Signals_47_2 AT %X47.2 : BOOL;
        Signals_47_3 AT %X47.3 : BOOL;
        Signals_47_4 AT %X47.4 : BOOL;
        Signals_47_5 AT %X47.5 : BOOL;
        Signals_47_6 AT %X47.6 : BOOL;
        Signals_47_7 AT %X47.7 : BOOL;
        Signals_48_0 AT %X48.0 : BOOL;
        Signals_48_1 AT %X48.1 : BOOL;
        Signals_48_2 AT %X48.2 : BOOL;
        Signals_48_3 AT %X48.3 : BOOL;
        Signals_48_4 AT %X48.4 : BOOL;
        Signals_48_5 AT %X48.5 : BOOL;
        Signals_48_6 AT %X48.6 : BOOL;
        Signals_48_7 AT %X48.7 : BOOL;
        Signals_49_0 AT %X49.0 : BOOL;
        Signals_49_1 AT %X49.1 : BOOL;
        Signals_49_2 AT %X49.2 : BOOL;
        Signals_49_3 AT %X49.3 : BOOL;
        Signals_49_4 AT %X49.4 : BOOL;
        Signals_49_5 AT %X49.5 : BOOL;
        Signals_49_6 AT %X49.6 : BOOL;
        Signals_49_7 AT %X49.7 : BOOL;
        Signals_50_0 AT %X50.0 : BOOL;
        Signals_50_1 AT %X50.1 : BOOL;
        Signals_50_2 AT %X50.2 : BOOL;
        Signals_50_3 AT %X50.3 : BOOL;
        Signals_50_4 AT %X50.4 : BOOL;
        Signals_50_5 AT %X50.5 : BOOL;
        Signals_50_6 AT %X50.6 : BOOL;
        Signals_50_7 AT %X50.7 : BOOL;
        Signals_51_0 AT %X51.0 : BOOL;
        Signals_51_1 AT %X51.1 : BOOL;
        Signals_51_2 AT %X51.2 : BOOL;
        Signals_51_3 AT %X51.3 : BOOL;
        Signals_51_4 AT %X51.4 : BOOL;
        Signals_51_5 AT %X51.5 : BOOL;
        Signals_51_6 AT %X51.6 : BOOL;
        Signals_51_7 AT %X51.7 : BOOL;
        Signals_52_0 AT %X52.0 : BOOL;
        Signals_52_1 AT %X52.1 : BOOL;
        Signals_52_2 AT %X52.2 : BOOL;
        Signals_52_3 AT %X52.3 : BOOL;
        Signals_52_4 AT %X52.4 : BOOL;
        Signals_52_5 AT %X52.5 : BOOL;
        Signals_52_6 AT %X52.6 : BOOL;
        Signals_52_7 AT %X52.7 : BOOL;
        Signals_53_0 AT %X53.0 : BOOL;
        Signals_53_1 AT %X53.1 : BOOL;
        Signals_53_2 AT %X53.2 : BOOL;
        Signals_53_3 AT %X53.3 : BOOL;
        Signals_53_4 AT %X53.4 : BOOL;
        Signals_53_5 AT %X53.5 : BOOL;
        Signals_53_6 AT %X53.6 : BOOL;
        Signals_53_7 AT %X53.7 : BOOL;
        Signals_54_0 AT %X54.0 : BOOL;
        Signals_54_1 AT %X54.1 : BOOL;
        Signals_54_2 AT %X54.2 : BOOL;
        Signals_54_3 AT %X54.3 : BOOL;
        Signals_54_4 AT %X54.4 : BOOL;
        Signals_54_5 AT %X54.5 : BOOL;
        Signals_54_6 AT %X54.6 : BOOL;
        Signals_54_7 AT %X54.7 : BOOL;
        Signals_55_0 AT %X55.0 : BOOL;
        Signals_55_1 AT %X55.1 : BOOL;
        Signals_55_2 AT %X55.2 : BOOL;
        Signals_55_3 AT %X55.3 : BOOL;
        Signals_55_4 AT %X55.4 : BOOL;
        Signals_55_5 AT %X55.5 : BOOL;
        Signals_55_6 AT %X55.6 : BOOL;
        Signals_55_7 AT %X55.7 : BOOL;
        Signals_56_0 AT %X56.0 : BOOL;
        Signals_56_1 AT %X56.1 : BOOL;
        Signals_56_2 AT %X56.2 : BOOL;
        Signals_56_3 AT %X56.3 : BOOL;
        Signals_56_4 AT %X56.4 : BOOL;
        Signals_56_5 AT %X56.5 : BOOL;
        Signals_56_6 AT %X56.6 : BOOL;
        Signals_56_7 AT %X56.7 : BOOL;
        Signals_57_0 AT %X57.0 : BOOL;
        Signals_57_1 AT %X57.1 : BOOL;
        Signals_57_2 AT %X57.2 : BOOL;
        Signals_57_3 AT %X57.3 : BOOL;
        Signals_57_4 AT %X57.4 : BOOL;
        Signals_57_5 AT %X57.5 : BOOL;
        Signals_57_6 AT %X57.6 : BOOL;
        Signals_57_7 AT %X57.7 : BOOL;
        Signals_58_0 AT %X58.0 : BOOL;
        Signals_58_1 AT %X58.1 : BOOL;
        Signals_58_2 AT %X58.2 : BOOL;
        Signals_58_3 AT %X58.3 : BOOL;
        Signals_58_4 AT %X58.4 : BOOL;
        Signals_58_5 AT %X58.5 : BOOL;
        Signals_58_6 AT %X58.6 : BOOL;
        Signals_58_7 AT %X58.7 : BOOL;
        Signals_59_0 AT %X59.0 : BOOL;
        Signals_59_1 AT %X59.1 : BOOL;
        Signals_59_2 AT %X59.2 : BOOL;
        Signals_59_3 AT %X59.3 : BOOL;
        Signals_59_4 AT %X59.4 : BOOL;
        Signals_59_5 AT %X59.5 : BOOL;
        Signals_59_6 AT %X59.6 : BOOL;
        Signals_59_7 AT %X59.7 : BOOL;
        Signals_60_0 AT %X60.0 : BOOL;
        Signals_60_1 AT %X60.1 : BOOL;
        Signals_60_2 AT %X60.2 : BOOL;
        Signals_60_3 AT %X60.3 : BOOL;
        Signals_60_4 AT %X60.4 : BOOL;
        Signals_60_5 AT %X60.5 : BOOL;
        Signals_60_6 AT %X60.6 : BOOL;
        Signals_60_7 AT %X60.7 : BOOL;
        Signals_61_0 AT %X61.0 : BOOL;
        Signals_61_1 AT %X61.1 : BOOL;
        Signals_61_2 AT %X61.2 : BOOL;
        Signals_61_3 AT %X61.3 : BOOL;
        Signals_61_4 AT %X61.4 : BOOL;
        Signals_61_5 AT %X61.5 : BOOL;
        Signals_61_6 AT %X61.6 : BOOL;
        Signals_61_7 AT %X61.7 : BOOL;
        Signals_62_0 AT %X62.0 : BOOL;
        Signals_62_1 AT %X62.1 : BOOL;
        Signals_62_2 AT %X62.2 : BOOL;
        Signals_62_3 AT %X62.3 : BOOL;
        Signals_62_4 AT %X62.4 : BOOL;
        Signals_62_5 AT %X62.5 : BOOL;
        Signals_62_6 AT %X62.6 : BOOL;
        Signals_62_7 AT %X62.7 : BOOL;
        Signals_63_0 AT %X63.0 : BOOL;
        Signals_63_1 AT %X63.1 : BOOL;
        Signals_63_2 AT %X63.2 : BOOL;
        Signals_63_3 AT %X63.3 : BOOL;
        Signals_63_4 AT %X63.4 : BOOL;
        Signals_63_5 AT %X63.5 : BOOL;
        Signals_63_6 AT %X63.6 : BOOL;
        Signals_63_7 AT %X63.7 : BOOL;
    END_STRUCT;
END_TYPE

TYPE
    kuka_rb2_DIO512_Output_Layout : STRUCT
        Signals_64_0 AT %X0.0 : BOOL;
        Signals_64_1 AT %X0.1 : BOOL;
        Signals_64_2 AT %X0.2 : BOOL;
        Signals_64_3 AT %X0.3 : BOOL;
        Signals_64_4 AT %X0.4 : BOOL;
        Signals_64_5 AT %X0.5 : BOOL;
        Signals_64_6 AT %X0.6 : BOOL;
        Signals_64_7 AT %X0.7 : BOOL;
        Signals_65_0 AT %X1.0 : BOOL;
        Signals_65_1 AT %X1.1 : BOOL;
        Signals_65_2 AT %X1.2 : BOOL;
        Signals_65_3 AT %X1.3 : BOOL;
        Signals_65_4 AT %X1.4 : BOOL;
        Signals_65_5 AT %X1.5 : BOOL;
        Signals_65_6 AT %X1.6 : BOOL;
        Signals_65_7 AT %X1.7 : BOOL;
        Signals_66_0 AT %X2.0 : BOOL;
        Signals_66_1 AT %X2.1 : BOOL;
        Signals_66_2 AT %X2.2 : BOOL;
        Signals_66_3 AT %X2.3 : BOOL;
        Signals_66_4 AT %X2.4 : BOOL;
        Signals_66_5 AT %X2.5 : BOOL;
        Signals_66_6 AT %X2.6 : BOOL;
        Signals_66_7 AT %X2.7 : BOOL;
        Signals_67_0 AT %X3.0 : BOOL;
        Signals_67_1 AT %X3.1 : BOOL;
        Signals_67_2 AT %X3.2 : BOOL;
        Signals_67_3 AT %X3.3 : BOOL;
        Signals_67_4 AT %X3.4 : BOOL;
        Signals_67_5 AT %X3.5 : BOOL;
        Signals_67_6 AT %X3.6 : BOOL;
        Signals_67_7 AT %X3.7 : BOOL;
        Signals_68_0 AT %X4.0 : BOOL;
        Signals_68_1 AT %X4.1 : BOOL;
        Signals_68_2 AT %X4.2 : BOOL;
        Signals_68_3 AT %X4.3 : BOOL;
        Signals_68_4 AT %X4.4 : BOOL;
        Signals_68_5 AT %X4.5 : BOOL;
        Signals_68_6 AT %X4.6 : BOOL;
        Signals_68_7 AT %X4.7 : BOOL;
        Signals_69_0 AT %X5.0 : BOOL;
        Signals_69_1 AT %X5.1 : BOOL;
        Signals_69_2 AT %X5.2 : BOOL;
        Signals_69_3 AT %X5.3 : BOOL;
        Signals_69_4 AT %X5.4 : BOOL;
        Signals_69_5 AT %X5.5 : BOOL;
        Signals_69_6 AT %X5.6 : BOOL;
        Signals_69_7 AT %X5.7 : BOOL;
        Signals_70_0 AT %X6.0 : BOOL;
        Signals_70_1 AT %X6.1 : BOOL;
        Signals_70_2 AT %X6.2 : BOOL;
        Signals_70_3 AT %X6.3 : BOOL;
        Signals_70_4 AT %X6.4 : BOOL;
        Signals_70_5 AT %X6.5 : BOOL;
        Signals_70_6 AT %X6.6 : BOOL;
        Signals_70_7 AT %X6.7 : BOOL;
        Signals_71_0 AT %X7.0 : BOOL;
        Signals_71_1 AT %X7.1 : BOOL;
        Signals_71_2 AT %X7.2 : BOOL;
        Signals_71_3 AT %X7.3 : BOOL;
        Signals_71_4 AT %X7.4 : BOOL;
        Signals_71_5 AT %X7.5 : BOOL;
        Signals_71_6 AT %X7.6 : BOOL;
        Signals_71_7 AT %X7.7 : BOOL;
        Signals_72_0 AT %X8.0 : BOOL;
        Signals_72_1 AT %X8.1 : BOOL;
        Signals_72_2 AT %X8.2 : BOOL;
        Signals_72_3 AT %X8.3 : BOOL;
        Signals_72_4 AT %X8.4 : BOOL;
        Signals_72_5 AT %X8.5 : BOOL;
        Signals_72_6 AT %X8.6 : BOOL;
        Signals_72_7 AT %X8.7 : BOOL;
        Signals_73_0 AT %X9.0 : BOOL;
        Signals_73_1 AT %X9.1 : BOOL;
        Signals_73_2 AT %X9.2 : BOOL;
        Signals_73_3 AT %X9.3 : BOOL;
        Signals_73_4 AT %X9.4 : BOOL;
        Signals_73_5 AT %X9.5 : BOOL;
        Signals_73_6 AT %X9.6 : BOOL;
        Signals_73_7 AT %X9.7 : BOOL;
        Signals_74_0 AT %X10.0 : BOOL;
        Signals_74_1 AT %X10.1 : BOOL;
        Signals_74_2 AT %X10.2 : BOOL;
        Signals_74_3 AT %X10.3 : BOOL;
        Signals_74_4 AT %X10.4 : BOOL;
        Signals_74_5 AT %X10.5 : BOOL;
        Signals_74_6 AT %X10.6 : BOOL;
        Signals_74_7 AT %X10.7 : BOOL;
        Signals_75_0 AT %X11.0 : BOOL;
        Signals_75_1 AT %X11.1 : BOOL;
        Signals_75_2 AT %X11.2 : BOOL;
        Signals_75_3 AT %X11.3 : BOOL;
        Signals_75_4 AT %X11.4 : BOOL;
        Signals_75_5 AT %X11.5 : BOOL;
        Signals_75_6 AT %X11.6 : BOOL;
        Signals_75_7 AT %X11.7 : BOOL;
        Signals_76_0 AT %X12.0 : BOOL;
        Signals_76_1 AT %X12.1 : BOOL;
        Signals_76_2 AT %X12.2 : BOOL;
        Signals_76_3 AT %X12.3 : BOOL;
        Signals_76_4 AT %X12.4 : BOOL;
        Signals_76_5 AT %X12.5 : BOOL;
        Signals_76_6 AT %X12.6 : BOOL;
        Signals_76_7 AT %X12.7 : BOOL;
        Signals_77_0 AT %X13.0 : BOOL;
        Signals_77_1 AT %X13.1 : BOOL;
        Signals_77_2 AT %X13.2 : BOOL;
        Signals_77_3 AT %X13.3 : BOOL;
        Signals_77_4 AT %X13.4 : BOOL;
        Signals_77_5 AT %X13.5 : BOOL;
        Signals_77_6 AT %X13.6 : BOOL;
        Signals_77_7 AT %X13.7 : BOOL;
        Signals_78_0 AT %X14.0 : BOOL;
        Signals_78_1 AT %X14.1 : BOOL;
        Signals_78_2 AT %X14.2 : BOOL;
        Signals_78_3 AT %X14.3 : BOOL;
        Signals_78_4 AT %X14.4 : BOOL;
        Signals_78_5 AT %X14.5 : BOOL;
        Signals_78_6 AT %X14.6 : BOOL;
        Signals_78_7 AT %X14.7 : BOOL;
        Signals_79_0 AT %X15.0 : BOOL;
        Signals_79_1 AT %X15.1 : BOOL;
        Signals_79_2 AT %X15.2 : BOOL;
        Signals_79_3 AT %X15.3 : BOOL;
        Signals_79_4 AT %X15.4 : BOOL;
        Signals_79_5 AT %X15.5 : BOOL;
        Signals_79_6 AT %X15.6 : BOOL;
        Signals_79_7 AT %X15.7 : BOOL;
        Signals_80_0 AT %X16.0 : BOOL;
        Signals_80_1 AT %X16.1 : BOOL;
        Signals_80_2 AT %X16.2 : BOOL;
        Signals_80_3 AT %X16.3 : BOOL;
        Signals_80_4 AT %X16.4 : BOOL;
        Signals_80_5 AT %X16.5 : BOOL;
        Signals_80_6 AT %X16.6 : BOOL;
        Signals_80_7 AT %X16.7 : BOOL;
        Signals_81_0 AT %X17.0 : BOOL;
        Signals_81_1 AT %X17.1 : BOOL;
        Signals_81_2 AT %X17.2 : BOOL;
        Signals_81_3 AT %X17.3 : BOOL;
        Signals_81_4 AT %X17.4 : BOOL;
        Signals_81_5 AT %X17.5 : BOOL;
        Signals_81_6 AT %X17.6 : BOOL;
        Signals_81_7 AT %X17.7 : BOOL;
        Signals_82_0 AT %X18.0 : BOOL;
        Signals_82_1 AT %X18.1 : BOOL;
        Signals_82_2 AT %X18.2 : BOOL;
        Signals_82_3 AT %X18.3 : BOOL;
        Signals_82_4 AT %X18.4 : BOOL;
        Signals_82_5 AT %X18.5 : BOOL;
        Signals_82_6 AT %X18.6 : BOOL;
        Signals_82_7 AT %X18.7 : BOOL;
        Signals_83_0 AT %X19.0 : BOOL;
        Signals_83_1 AT %X19.1 : BOOL;
        Signals_83_2 AT %X19.2 : BOOL;
        Signals_83_3 AT %X19.3 : BOOL;
        Signals_83_4 AT %X19.4 : BOOL;
        Signals_83_5 AT %X19.5 : BOOL;
        Signals_83_6 AT %X19.6 : BOOL;
        Signals_83_7 AT %X19.7 : BOOL;
        Signals_84_0 AT %X20.0 : BOOL;
        Signals_84_1 AT %X20.1 : BOOL;
        Signals_84_2 AT %X20.2 : BOOL;
        Signals_84_3 AT %X20.3 : BOOL;
        Signals_84_4 AT %X20.4 : BOOL;
        Signals_84_5 AT %X20.5 : BOOL;
        Signals_84_6 AT %X20.6 : BOOL;
        Signals_84_7 AT %X20.7 : BOOL;
        Signals_85_0 AT %X21.0 : BOOL;
        Signals_85_1 AT %X21.1 : BOOL;
        Signals_85_2 AT %X21.2 : BOOL;
        Signals_85_3 AT %X21.3 : BOOL;
        Signals_85_4 AT %X21.4 : BOOL;
        Signals_85_5 AT %X21.5 : BOOL;
        Signals_85_6 AT %X21.6 : BOOL;
        Signals_85_7 AT %X21.7 : BOOL;
        Signals_86_0 AT %X22.0 : BOOL;
        Signals_86_1 AT %X22.1 : BOOL;
        Signals_86_2 AT %X22.2 : BOOL;
        Signals_86_3 AT %X22.3 : BOOL;
        Signals_86_4 AT %X22.4 : BOOL;
        Signals_86_5 AT %X22.5 : BOOL;
        Signals_86_6 AT %X22.6 : BOOL;
        Signals_86_7 AT %X22.7 : BOOL;
        Signals_87_0 AT %X23.0 : BOOL;
        Signals_87_1 AT %X23.1 : BOOL;
        Signals_87_2 AT %X23.2 : BOOL;
        Signals_87_3 AT %X23.3 : BOOL;
        Signals_87_4 AT %X23.4 : BOOL;
        Signals_87_5 AT %X23.5 : BOOL;
        Signals_87_6 AT %X23.6 : BOOL;
        Signals_87_7 AT %X23.7 : BOOL;
        Signals_88_0 AT %X24.0 : BOOL;
        Signals_88_1 AT %X24.1 : BOOL;
        Signals_88_2 AT %X24.2 : BOOL;
        Signals_88_3 AT %X24.3 : BOOL;
        Signals_88_4 AT %X24.4 : BOOL;
        Signals_88_5 AT %X24.5 : BOOL;
        Signals_88_6 AT %X24.6 : BOOL;
        Signals_88_7 AT %X24.7 : BOOL;
        Signals_89_0 AT %X25.0 : BOOL;
        Signals_89_1 AT %X25.1 : BOOL;
        Signals_89_2 AT %X25.2 : BOOL;
        Signals_89_3 AT %X25.3 : BOOL;
        Signals_89_4 AT %X25.4 : BOOL;
        Signals_89_5 AT %X25.5 : BOOL;
        Signals_89_6 AT %X25.6 : BOOL;
        Signals_89_7 AT %X25.7 : BOOL;
        Signals_90_0 AT %X26.0 : BOOL;
        Signals_90_1 AT %X26.1 : BOOL;
        Signals_90_2 AT %X26.2 : BOOL;
        Signals_90_3 AT %X26.3 : BOOL;
        Signals_90_4 AT %X26.4 : BOOL;
        Signals_90_5 AT %X26.5 : BOOL;
        Signals_90_6 AT %X26.6 : BOOL;
        Signals_90_7 AT %X26.7 : BOOL;
        Signals_91_0 AT %X27.0 : BOOL;
        Signals_91_1 AT %X27.1 : BOOL;
        Signals_91_2 AT %X27.2 : BOOL;
        Signals_91_3 AT %X27.3 : BOOL;
        Signals_91_4 AT %X27.4 : BOOL;
        Signals_91_5 AT %X27.5 : BOOL;
        Signals_91_6 AT %X27.6 : BOOL;
        Signals_91_7 AT %X27.7 : BOOL;
        Signals_92_0 AT %X28.0 : BOOL;
        Signals_92_1 AT %X28.1 : BOOL;
        Signals_92_2 AT %X28.2 : BOOL;
        Signals_92_3 AT %X28.3 : BOOL;
        Signals_92_4 AT %X28.4 : BOOL;
        Signals_92_5 AT %X28.5 : BOOL;
        Signals_92_6 AT %X28.6 : BOOL;
        Signals_92_7 AT %X28.7 : BOOL;
        Signals_93_0 AT %X29.0 : BOOL;
        Signals_93_1 AT %X29.1 : BOOL;
        Signals_93_2 AT %X29.2 : BOOL;
        Signals_93_3 AT %X29.3 : BOOL;
        Signals_93_4 AT %X29.4 : BOOL;
        Signals_93_5 AT %X29.5 : BOOL;
        Signals_93_6 AT %X29.6 : BOOL;
        Signals_93_7 AT %X29.7 : BOOL;
        Signals_94_0 AT %X30.0 : BOOL;
        Signals_94_1 AT %X30.1 : BOOL;
        Signals_94_2 AT %X30.2 : BOOL;
        Signals_94_3 AT %X30.3 : BOOL;
        Signals_94_4 AT %X30.4 : BOOL;
        Signals_94_5 AT %X30.5 : BOOL;
        Signals_94_6 AT %X30.6 : BOOL;
        Signals_94_7 AT %X30.7 : BOOL;
        Signals_95_0 AT %X31.0 : BOOL;
        Signals_95_1 AT %X31.1 : BOOL;
        Signals_95_2 AT %X31.2 : BOOL;
        Signals_95_3 AT %X31.3 : BOOL;
        Signals_95_4 AT %X31.4 : BOOL;
        Signals_95_5 AT %X31.5 : BOOL;
        Signals_95_6 AT %X31.6 : BOOL;
        Signals_95_7 AT %X31.7 : BOOL;
        Signals_96_0 AT %X32.0 : BOOL;
        Signals_96_1 AT %X32.1 : BOOL;
        Signals_96_2 AT %X32.2 : BOOL;
        Signals_96_3 AT %X32.3 : BOOL;
        Signals_96_4 AT %X32.4 : BOOL;
        Signals_96_5 AT %X32.5 : BOOL;
        Signals_96_6 AT %X32.6 : BOOL;
        Signals_96_7 AT %X32.7 : BOOL;
        Signals_97_0 AT %X33.0 : BOOL;
        Signals_97_1 AT %X33.1 : BOOL;
        Signals_97_2 AT %X33.2 : BOOL;
        Signals_97_3 AT %X33.3 : BOOL;
        Signals_97_4 AT %X33.4 : BOOL;
        Signals_97_5 AT %X33.5 : BOOL;
        Signals_97_6 AT %X33.6 : BOOL;
        Signals_97_7 AT %X33.7 : BOOL;
        Signals_98_0 AT %X34.0 : BOOL;
        Signals_98_1 AT %X34.1 : BOOL;
        Signals_98_2 AT %X34.2 : BOOL;
        Signals_98_3 AT %X34.3 : BOOL;
        Signals_98_4 AT %X34.4 : BOOL;
        Signals_98_5 AT %X34.5 : BOOL;
        Signals_98_6 AT %X34.6 : BOOL;
        Signals_98_7 AT %X34.7 : BOOL;
        Signals_99_0 AT %X35.0 : BOOL;
        Signals_99_1 AT %X35.1 : BOOL;
        Signals_99_2 AT %X35.2 : BOOL;
        Signals_99_3 AT %X35.3 : BOOL;
        Signals_99_4 AT %X35.4 : BOOL;
        Signals_99_5 AT %X35.5 : BOOL;
        Signals_99_6 AT %X35.6 : BOOL;
        Signals_99_7 AT %X35.7 : BOOL;
        Signals_100_0 AT %X36.0 : BOOL;
        Signals_100_1 AT %X36.1 : BOOL;
        Signals_100_2 AT %X36.2 : BOOL;
        Signals_100_3 AT %X36.3 : BOOL;
        Signals_100_4 AT %X36.4 : BOOL;
        Signals_100_5 AT %X36.5 : BOOL;
        Signals_100_6 AT %X36.6 : BOOL;
        Signals_100_7 AT %X36.7 : BOOL;
        Signals_101_0 AT %X37.0 : BOOL;
        Signals_101_1 AT %X37.1 : BOOL;
        Signals_101_2 AT %X37.2 : BOOL;
        Signals_101_3 AT %X37.3 : BOOL;
        Signals_101_4 AT %X37.4 : BOOL;
        Signals_101_5 AT %X37.5 : BOOL;
        Signals_101_6 AT %X37.6 : BOOL;
        Signals_101_7 AT %X37.7 : BOOL;
        Signals_102_0 AT %X38.0 : BOOL;
        Signals_102_1 AT %X38.1 : BOOL;
        Signals_102_2 AT %X38.2 : BOOL;
        Signals_102_3 AT %X38.3 : BOOL;
        Signals_102_4 AT %X38.4 : BOOL;
        Signals_102_5 AT %X38.5 : BOOL;
        Signals_102_6 AT %X38.6 : BOOL;
        Signals_102_7 AT %X38.7 : BOOL;
        Signals_103_0 AT %X39.0 : BOOL;
        Signals_103_1 AT %X39.1 : BOOL;
        Signals_103_2 AT %X39.2 : BOOL;
        Signals_103_3 AT %X39.3 : BOOL;
        Signals_103_4 AT %X39.4 : BOOL;
        Signals_103_5 AT %X39.5 : BOOL;
        Signals_103_6 AT %X39.6 : BOOL;
        Signals_103_7 AT %X39.7 : BOOL;
        Signals_104_0 AT %X40.0 : BOOL;
        Signals_104_1 AT %X40.1 : BOOL;
        Signals_104_2 AT %X40.2 : BOOL;
        Signals_104_3 AT %X40.3 : BOOL;
        Signals_104_4 AT %X40.4 : BOOL;
        Signals_104_5 AT %X40.5 : BOOL;
        Signals_104_6 AT %X40.6 : BOOL;
        Signals_104_7 AT %X40.7 : BOOL;
        Signals_105_0 AT %X41.0 : BOOL;
        Signals_105_1 AT %X41.1 : BOOL;
        Signals_105_2 AT %X41.2 : BOOL;
        Signals_105_3 AT %X41.3 : BOOL;
        Signals_105_4 AT %X41.4 : BOOL;
        Signals_105_5 AT %X41.5 : BOOL;
        Signals_105_6 AT %X41.6 : BOOL;
        Signals_105_7 AT %X41.7 : BOOL;
        Signals_106_0 AT %X42.0 : BOOL;
        Signals_106_1 AT %X42.1 : BOOL;
        Signals_106_2 AT %X42.2 : BOOL;
        Signals_106_3 AT %X42.3 : BOOL;
        Signals_106_4 AT %X42.4 : BOOL;
        Signals_106_5 AT %X42.5 : BOOL;
        Signals_106_6 AT %X42.6 : BOOL;
        Signals_106_7 AT %X42.7 : BOOL;
        Signals_107_0 AT %X43.0 : BOOL;
        Signals_107_1 AT %X43.1 : BOOL;
        Signals_107_2 AT %X43.2 : BOOL;
        Signals_107_3 AT %X43.3 : BOOL;
        Signals_107_4 AT %X43.4 : BOOL;
        Signals_107_5 AT %X43.5 : BOOL;
        Signals_107_6 AT %X43.6 : BOOL;
        Signals_107_7 AT %X43.7 : BOOL;
        Signals_108_0 AT %X44.0 : BOOL;
        Signals_108_1 AT %X44.1 : BOOL;
        Signals_108_2 AT %X44.2 : BOOL;
        Signals_108_3 AT %X44.3 : BOOL;
        Signals_108_4 AT %X44.4 : BOOL;
        Signals_108_5 AT %X44.5 : BOOL;
        Signals_108_6 AT %X44.6 : BOOL;
        Signals_108_7 AT %X44.7 : BOOL;
        Signals_109_0 AT %X45.0 : BOOL;
        Signals_109_1 AT %X45.1 : BOOL;
        Signals_109_2 AT %X45.2 : BOOL;
        Signals_109_3 AT %X45.3 : BOOL;
        Signals_109_4 AT %X45.4 : BOOL;
        Signals_109_5 AT %X45.5 : BOOL;
        Signals_109_6 AT %X45.6 : BOOL;
        Signals_109_7 AT %X45.7 : BOOL;
        Signals_110_0 AT %X46.0 : BOOL;
        Signals_110_1 AT %X46.1 : BOOL;
        Signals_110_2 AT %X46.2 : BOOL;
        Signals_110_3 AT %X46.3 : BOOL;
        Signals_110_4 AT %X46.4 : BOOL;
        Signals_110_5 AT %X46.5 : BOOL;
        Signals_110_6 AT %X46.6 : BOOL;
        Signals_110_7 AT %X46.7 : BOOL;
        Signals_111_0 AT %X47.0 : BOOL;
        Signals_111_1 AT %X47.1 : BOOL;
        Signals_111_2 AT %X47.2 : BOOL;
        Signals_111_3 AT %X47.3 : BOOL;
        Signals_111_4 AT %X47.4 : BOOL;
        Signals_111_5 AT %X47.5 : BOOL;
        Signals_111_6 AT %X47.6 : BOOL;
        Signals_111_7 AT %X47.7 : BOOL;
        Signals_112_0 AT %X48.0 : BOOL;
        Signals_112_1 AT %X48.1 : BOOL;
        Signals_112_2 AT %X48.2 : BOOL;
        Signals_112_3 AT %X48.3 : BOOL;
        Signals_112_4 AT %X48.4 : BOOL;
        Signals_112_5 AT %X48.5 : BOOL;
        Signals_112_6 AT %X48.6 : BOOL;
        Signals_112_7 AT %X48.7 : BOOL;
        Signals_113_0 AT %X49.0 : BOOL;
        Signals_113_1 AT %X49.1 : BOOL;
        Signals_113_2 AT %X49.2 : BOOL;
        Signals_113_3 AT %X49.3 : BOOL;
        Signals_113_4 AT %X49.4 : BOOL;
        Signals_113_5 AT %X49.5 : BOOL;
        Signals_113_6 AT %X49.6 : BOOL;
        Signals_113_7 AT %X49.7 : BOOL;
        Signals_114_0 AT %X50.0 : BOOL;
        Signals_114_1 AT %X50.1 : BOOL;
        Signals_114_2 AT %X50.2 : BOOL;
        Signals_114_3 AT %X50.3 : BOOL;
        Signals_114_4 AT %X50.4 : BOOL;
        Signals_114_5 AT %X50.5 : BOOL;
        Signals_114_6 AT %X50.6 : BOOL;
        Signals_114_7 AT %X50.7 : BOOL;
        Signals_115_0 AT %X51.0 : BOOL;
        Signals_115_1 AT %X51.1 : BOOL;
        Signals_115_2 AT %X51.2 : BOOL;
        Signals_115_3 AT %X51.3 : BOOL;
        Signals_115_4 AT %X51.4 : BOOL;
        Signals_115_5 AT %X51.5 : BOOL;
        Signals_115_6 AT %X51.6 : BOOL;
        Signals_115_7 AT %X51.7 : BOOL;
        Signals_116_0 AT %X52.0 : BOOL;
        Signals_116_1 AT %X52.1 : BOOL;
        Signals_116_2 AT %X52.2 : BOOL;
        Signals_116_3 AT %X52.3 : BOOL;
        Signals_116_4 AT %X52.4 : BOOL;
        Signals_116_5 AT %X52.5 : BOOL;
        Signals_116_6 AT %X52.6 : BOOL;
        Signals_116_7 AT %X52.7 : BOOL;
        Signals_117_0 AT %X53.0 : BOOL;
        Signals_117_1 AT %X53.1 : BOOL;
        Signals_117_2 AT %X53.2 : BOOL;
        Signals_117_3 AT %X53.3 : BOOL;
        Signals_117_4 AT %X53.4 : BOOL;
        Signals_117_5 AT %X53.5 : BOOL;
        Signals_117_6 AT %X53.6 : BOOL;
        Signals_117_7 AT %X53.7 : BOOL;
        Signals_118_0 AT %X54.0 : BOOL;
        Signals_118_1 AT %X54.1 : BOOL;
        Signals_118_2 AT %X54.2 : BOOL;
        Signals_118_3 AT %X54.3 : BOOL;
        Signals_118_4 AT %X54.4 : BOOL;
        Signals_118_5 AT %X54.5 : BOOL;
        Signals_118_6 AT %X54.6 : BOOL;
        Signals_118_7 AT %X54.7 : BOOL;
        Signals_119_0 AT %X55.0 : BOOL;
        Signals_119_1 AT %X55.1 : BOOL;
        Signals_119_2 AT %X55.2 : BOOL;
        Signals_119_3 AT %X55.3 : BOOL;
        Signals_119_4 AT %X55.4 : BOOL;
        Signals_119_5 AT %X55.5 : BOOL;
        Signals_119_6 AT %X55.6 : BOOL;
        Signals_119_7 AT %X55.7 : BOOL;
        Signals_120_0 AT %X56.0 : BOOL;
        Signals_120_1 AT %X56.1 : BOOL;
        Signals_120_2 AT %X56.2 : BOOL;
        Signals_120_3 AT %X56.3 : BOOL;
        Signals_120_4 AT %X56.4 : BOOL;
        Signals_120_5 AT %X56.5 : BOOL;
        Signals_120_6 AT %X56.6 : BOOL;
        Signals_120_7 AT %X56.7 : BOOL;
        Signals_121_0 AT %X57.0 : BOOL;
        Signals_121_1 AT %X57.1 : BOOL;
        Signals_121_2 AT %X57.2 : BOOL;
        Signals_121_3 AT %X57.3 : BOOL;
        Signals_121_4 AT %X57.4 : BOOL;
        Signals_121_5 AT %X57.5 : BOOL;
        Signals_121_6 AT %X57.6 : BOOL;
        Signals_121_7 AT %X57.7 : BOOL;
        Signals_122_0 AT %X58.0 : BOOL;
        Signals_122_1 AT %X58.1 : BOOL;
        Signals_122_2 AT %X58.2 : BOOL;
        Signals_122_3 AT %X58.3 : BOOL;
        Signals_122_4 AT %X58.4 : BOOL;
        Signals_122_5 AT %X58.5 : BOOL;
        Signals_122_6 AT %X58.6 : BOOL;
        Signals_122_7 AT %X58.7 : BOOL;
        Signals_123_0 AT %X59.0 : BOOL;
        Signals_123_1 AT %X59.1 : BOOL;
        Signals_123_2 AT %X59.2 : BOOL;
        Signals_123_3 AT %X59.3 : BOOL;
        Signals_123_4 AT %X59.4 : BOOL;
        Signals_123_5 AT %X59.5 : BOOL;
        Signals_123_6 AT %X59.6 : BOOL;
        Signals_123_7 AT %X59.7 : BOOL;
        Signals_124_0 AT %X60.0 : BOOL;
        Signals_124_1 AT %X60.1 : BOOL;
        Signals_124_2 AT %X60.2 : BOOL;
        Signals_124_3 AT %X60.3 : BOOL;
        Signals_124_4 AT %X60.4 : BOOL;
        Signals_124_5 AT %X60.5 : BOOL;
        Signals_124_6 AT %X60.6 : BOOL;
        Signals_124_7 AT %X60.7 : BOOL;
        Signals_125_0 AT %X61.0 : BOOL;
        Signals_125_1 AT %X61.1 : BOOL;
        Signals_125_2 AT %X61.2 : BOOL;
        Signals_125_3 AT %X61.3 : BOOL;
        Signals_125_4 AT %X61.4 : BOOL;
        Signals_125_5 AT %X61.5 : BOOL;
        Signals_125_6 AT %X61.6 : BOOL;
        Signals_125_7 AT %X61.7 : BOOL;
        Signals_126_0 AT %X62.0 : BOOL;
        Signals_126_1 AT %X62.1 : BOOL;
        Signals_126_2 AT %X62.2 : BOOL;
        Signals_126_3 AT %X62.3 : BOOL;
        Signals_126_4 AT %X62.4 : BOOL;
        Signals_126_5 AT %X62.5 : BOOL;
        Signals_126_6 AT %X62.6 : BOOL;
        Signals_126_7 AT %X62.7 : BOOL;
        Signals_127_0 AT %X63.0 : BOOL;
        Signals_127_1 AT %X63.1 : BOOL;
        Signals_127_2 AT %X63.2 : BOOL;
        Signals_127_3 AT %X63.3 : BOOL;
        Signals_127_4 AT %X63.4 : BOOL;
        Signals_127_5 AT %X63.5 : BOOL;
        Signals_127_6 AT %X63.6 : BOOL;
        Signals_127_7 AT %X63.7 : BOOL;
    END_STRUCT;
END_TYPE

TYPE
    mitsubishi_tz535_robot_In_Out_64_byte_Input_Layout : STRUCT
        Signals_0 AT %B0 : ARRAY[0..63] OF BYTE;
    END_STRUCT;
END_TYPE

TYPE
    mitsubishi_tz535_robot_In_Out_64_byte_Output_Layout : STRUCT
        Signals_1 AT %B0 : ARRAY[0..63] OF BYTE;
    END_STRUCT;
END_TYPE

TYPE
    plc_line_A1_Input_Layout : STRUCT
        Channel_00DI AT %X0.0 : BOOL;
        Channel_01DI AT %X0.1 : BOOL;
        Channel_02DI AT %X0.2 : BOOL;
        Channel_03DI AT %X0.3 : BOOL;
        Channel_04DI AT %X0.4 : BOOL;
        Channel_05DI AT %X0.5 : BOOL;
        Channel_06DI AT %X0.6 : BOOL;
        Channel_07DI AT %X0.7 : BOOL;
        Channel_08DI AT %X1.0 : BOOL;
        Channel_09DI AT %X1.1 : BOOL;
        Channel_10DI AT %X1.2 : BOOL;
        Channel_11DI AT %X1.3 : BOOL;
        Channel_12DI AT %X1.4 : BOOL;
        Channel_13DI AT %X1.5 : BOOL;
        Channel_14DI AT %X1.6 : BOOL;
        Channel_15DI AT %X1.7 : BOOL;
        Channel_16DI AT %X2.0 : BOOL;
        Channel_17DI AT %X2.1 : BOOL;
        Channel_18DI AT %X2.2 : BOOL;
        Channel_19DI AT %X2.3 : BOOL;
        Channel_20DI AT %X2.4 : BOOL;
        Channel_21DI AT %X2.5 : BOOL;
        Channel_22DI AT %X2.6 : BOOL;
        Channel_23DI AT %X2.7 : BOOL;
        Channel_24DI AT %X3.0 : BOOL;
        Channel_25DI AT %X3.1 : BOOL;
        Channel_26DI AT %X3.2 : BOOL;
        Channel_27DI AT %X3.3 : BOOL;
        Channel_28DI AT %X3.4 : BOOL;
        Channel_29DI AT %X3.5 : BOOL;
        Channel_30DI AT %X3.6 : BOOL;
        Channel_31DI AT %X3.7 : BOOL;
    END_STRUCT;
END_TYPE

TYPE
    rexroth_cs351_Input_2_word_1_Input_Layout : STRUCT
        Signals_0 AT %B0 : DWORD;
    END_STRUCT;
END_TYPE

TYPE
    rexroth_cs351_Input_4_word_1_Input_Layout : STRUCT
        Signals_0 AT %B0 : DWORD;
        Signals_1 AT %B4 : DWORD;
    END_STRUCT;
END_TYPE

TYPE
    rexroth_cs351_Input_4_word_10_Input_Layout : STRUCT
        Signals_0 AT %B0 : DWORD;
        Signals_1 AT %B4 : DWORD;
    END_STRUCT;
END_TYPE

TYPE
    rexroth_cs351_Input_4_word_11_Input_Layout : STRUCT
        Signals_0 AT %B0 : DWORD;
        Signals_1 AT %B4 : DWORD;
    END_STRUCT;
END_TYPE

TYPE
    rexroth_cs351_Input_4_word_12_Input_Layout : STRUCT
        Signals_0 AT %B0 : DWORD;
        Signals_1 AT %B4 : DWORD;
    END_STRUCT;
END_TYPE

TYPE
    rexroth_cs351_Input_4_word_13_Input_Layout : STRUCT
        Signals_0 AT %B0 : DWORD;
        Signals_1 AT %B4 : DWORD;
    END_STRUCT;
END_TYPE

TYPE
    rexroth_cs351_Input_4_word_14_Input_Layout : STRUCT
        Signals_0 AT %B0 : DWORD;
        Signals_1 AT %B4 : DWORD;
    END_STRUCT;
END_TYPE

TYPE
    rexroth_cs351_Input_4_word_15_Input_Layout : STRUCT
        Signals_0 AT %B0 : DWORD;
        Signals_1 AT %B4 : DWORD;
    END_STRUCT;
END_TYPE

TYPE
    rexroth_cs351_Input_4_word_16_Input_Layout : STRUCT
        Signals_0 AT %B0 : DWORD;
        Signals_1 AT %B4 : DWORD;
    END_STRUCT;
END_TYPE

TYPE
    rexroth_cs351_Input_4_word_2_Input_Layout : STRUCT
        Signals_0 AT %B0 : DWORD;
        Signals_1 AT %B4 : DWORD;
    END_STRUCT;
END_TYPE

TYPE
    rexroth_cs351_Input_4_word_3_Input_Layout : STRUCT
        Signals_0 AT %B0 : DWORD;
        Signals_1 AT %B4 : DWORD;
    END_STRUCT;
END_TYPE

TYPE
    rexroth_cs351_Input_4_word_4_Input_Layout : STRUCT
        Signals_0 AT %B0 : DWORD;
        Signals_1 AT %B4 : DWORD;
    END_STRUCT;
END_TYPE

TYPE
    rexroth_cs351_Input_4_word_5_Input_Layout : STRUCT
        Signals_0 AT %B0 : DWORD;
        Signals_1 AT %B4 : DWORD;
    END_STRUCT;
END_TYPE

TYPE
    rexroth_cs351_Input_4_word_6_Input_Layout : STRUCT
        Signals_0 AT %B0 : DWORD;
        Signals_1 AT %B4 : DWORD;
    END_STRUCT;
END_TYPE

TYPE
    rexroth_cs351_Input_4_word_7_Input_Layout : STRUCT
        Signals_0 AT %B0 : DWORD;
        Signals_1 AT %B4 : DWORD;
    END_STRUCT;
END_TYPE

TYPE
    rexroth_cs351_Input_4_word_8_Input_Layout : STRUCT
        Signals_0 AT %B0 : DWORD;
        Signals_1 AT %B4 : DWORD;
    END_STRUCT;
END_TYPE

TYPE
    rexroth_cs351_Input_4_word_9_Input_Layout : STRUCT
        Signals_0 AT %B0 : DWORD;
        Signals_1 AT %B4 : DWORD;
    END_STRUCT;
END_TYPE

TYPE
    rexroth_cs351_Output_2_word_1_Output_Layout : STRUCT
        Signals_0 AT %B0 : DWORD;
    END_STRUCT;
END_TYPE

TYPE
    rexroth_cs351_Output_4_word_1_Output_Layout : STRUCT
        Signals_0 AT %B0 : DWORD;
        Signals_1 AT %B4 : DWORD;
    END_STRUCT;
END_TYPE

TYPE
    rexroth_cs351_Output_4_word_2_Output_Layout : STRUCT
        Signals_0 AT %B0 : DWORD;
        Signals_1 AT %B4 : DWORD;
    END_STRUCT;
END_TYPE

TYPE
    rexroth_cs351_Output_4_word_3_Output_Layout : STRUCT
        Signals_0 AT %B0 : DWORD;
        Signals_1 AT %B4 : DWORD;
    END_STRUCT;
END_TYPE

TYPE
    rexroth_cs351_Output_4_word_4_Output_Layout : STRUCT
        Signals_0 AT %B0 : DWORD;
        Signals_1 AT %B4 : DWORD;
    END_STRUCT;
END_TYPE

TYPE
    rexroth_cs351_Output_4_word_5_Output_Layout : STRUCT
        Signals_0 AT %B0 : DWORD;
        Signals_1 AT %B4 : DWORD;
    END_STRUCT;
END_TYPE

TYPE
    rexroth_cs351_Output_4_word_6_Output_Layout : STRUCT
        Signals_0 AT %B0 : DWORD;
        Signals_1 AT %B4 : DWORD;
    END_STRUCT;
END_TYPE

TYPE
    rexroth_cs351_Output_4_word_7_Output_Layout : STRUCT
        Signals_0 AT %B0 : DWORD;
        Signals_1 AT %B4 : DWORD;
    END_STRUCT;
END_TYPE

TYPE
    rexroth_cs351_Output_4_word_8_Output_Layout : STRUCT
        Signals_0 AT %B0 : DWORD;
        Signals_1 AT %B4 : DWORD;
    END_STRUCT;
END_TYPE

TYPE
    rexroth_ctrlx_drive_Inputs_P_0_0106_0_0__STO_function__Operating_status_Input_Layout : STRUCT
        Signals_0 AT %B0 : WORD;
    END_STRUCT;
END_TYPE

TYPE
    rexroth_ctrlx_drive_Inputs_S_0_0084_0_0__Torque_force_feedback_value_Input_Layout : STRUCT
        Signals_0 AT %B0 : INT;
    END_STRUCT;
END_TYPE

TYPE
    rexroth_ctrlx_drive_Inputs_S_0_0135_0_0__Drive_status_word__Value_Input_Layout : STRUCT
        Signals_0 AT %X0.3 : BOOL;
        Signals_1 AT %X0.4 : BOOL;
        Signals_2 AT %X0.5 : BOOL;
        Signals_3 AT %X0.7 : BOOL;
        Signals_4 AT %X1.0 : BOOL;
        Signals_5 AT %X1.1 : BOOL;
        Signals_6 AT %X1.2 : BOOL;
        Signals_7 AT %X1.4 : BOOL;
        Signals_8 AT %X1.5 : BOOL;
        Signals_9 AT %X1.6 : BOOL;
        Signals_10 AT %X1.7 : BOOL;
    END_STRUCT;
END_TYPE

TYPE
    rexroth_ctrlx_drive_Inputs_S_0_0144_0_0__Signal_status_word__Value_Input_Layout : STRUCT
        Signals_0 AT %B0 : WORD;
    END_STRUCT;
END_TYPE

TYPE
    rexroth_ctrlx_drive_Inputs_S_0_0386_0_0__Position_controller__Position_actual_value_Input_Layout : STRUCT
        Signals_0 AT %B0 : DINT;
    END_STRUCT;
END_TYPE

TYPE
    rexroth_ctrlx_drive_Inputs_S_0_0390_0_0__Diagnostic_message__Manufacturer_status_register_Input_Layout : STRUCT
        Signals_0 AT %B0 : DWORD;
    END_STRUCT;
END_TYPE

TYPE
    rexroth_ctrlx_drive_Inputs_S_0_0535_0_0__Velocity_controller__Velocity_actual_value_Input_Layout : STRUCT
        Signals_0 AT %B0 : DINT;
    END_STRUCT;
END_TYPE

TYPE
    rexroth_ctrlx_drive_Inputs_S_0_1720_0_2__Power_supply_control__Status_word_Input_Layout : STRUCT
        Signals_0 AT %B0 : WORD;
    END_STRUCT;
END_TYPE

TYPE
    rexroth_ctrlx_drive_Outputs_S_0_0080_0_0__Torque_force_command_value_Output_Layout : STRUCT
        Signals_0 AT %B0 : INT;
    END_STRUCT;
END_TYPE

TYPE
    rexroth_ctrlx_drive_Outputs_S_0_0092_0_0__Torque_force_limitation__Limit_value_bipolar_Output_Layout : STRUCT
        Signals_0 AT %B0 : WORD;
    END_STRUCT;
END_TYPE

TYPE
    rexroth_ctrlx_drive_Outputs_S_0_0134_0_0__Master_control_word__Value_Output_Layout : STRUCT
        Signals_0 AT %X1.0 : BOOL;
        Signals_1 AT %X1.1 : BOOL;
        Signals_2 AT %X1.2 : BOOL;
        Signals_3 AT %X1.5 : BOOL;
        Signals_4 AT %X1.6 : BOOL;
        Signals_5 AT %X1.7 : BOOL;
    END_STRUCT;
END_TYPE

TYPE
    rexroth_ctrlx_drive_Outputs_S_0_0145_0_0__Signal_control_word__Value_Output_Layout : STRUCT
        Signals_0 AT %B0 : WORD;
    END_STRUCT;
END_TYPE

TYPE
    rexroth_ctrlx_drive_Outputs_S_0_0193_0_0__Positioning_jerk_Output_Layout : STRUCT
        Signals_0 AT %B0 : DINT;
    END_STRUCT;
END_TYPE

TYPE
    rexroth_ctrlx_drive_Outputs_S_0_0259_0_0__Positioning_profile__Profile_velocity_Output_Layout : STRUCT
        Signals_0 AT %B0 : DWORD;
    END_STRUCT;
END_TYPE

TYPE
    rexroth_ctrlx_drive_Outputs_S_0_0260_0_0__Positioning_profile__Acceleration_Output_Layout : STRUCT
        Signals_0 AT %B0 : DINT;
    END_STRUCT;
END_TYPE

TYPE
    rexroth_ctrlx_drive_Outputs_S_0_0282_0_0__Drive_controlled_positioning__Command_value_Output_Layout : STRUCT
        Signals_0 AT %B0 : DINT;
    END_STRUCT;
END_TYPE

TYPE
    rexroth_ctrlx_drive_Outputs_S_0_0359_0_0__Positioning_profile__Deceleration_Output_Layout : STRUCT
        Signals_0 AT %B0 : DINT;
    END_STRUCT;
END_TYPE

TYPE
    rexroth_ctrlx_drive_Outputs_S_0_1720_0_1__Power_supply_control__Control_word_Output_Layout : STRUCT
        Signals_0 AT %B0 : WORD;
    END_STRUCT;
END_TYPE

TYPE
    rexroth_indradrive_Input_9_Words_Input_Layout : STRUCT
        Signals_0 AT %B0 : WORD;
        Signals_1 AT %B2 : WORD;
        Signals_2 AT %B4 : WORD;
        Signals_3 AT %B6 : WORD;
        Signals_4 AT %B8 : WORD;
        Signals_5 AT %B10 : WORD;
        Signals_6 AT %B12 : WORD;
        Signals_7 AT %B14 : WORD;
        Signals_8 AT %B16 : WORD;
    END_STRUCT;
END_TYPE

TYPE
    rexroth_indradrive_Output_13_Words_Output_Layout : STRUCT
        Signals_0 AT %B0 : WORD;
        Signals_1 AT %B2 : WORD;
        Signals_2 AT %B4 : WORD;
        Signals_3 AT %B6 : WORD;
        Signals_4 AT %B8 : WORD;
        Signals_5 AT %B10 : WORD;
        Signals_6 AT %B12 : WORD;
        Signals_7 AT %B14 : WORD;
        Signals_8 AT %B16 : WORD;
        Signals_9 AT %B18 : WORD;
        Signals_10 AT %B20 : WORD;
        Signals_11 AT %B22 : WORD;
        Signals_12 AT %B24 : WORD;
    END_STRUCT;
END_TYPE

TYPE
    rexroth_indradrive_ParamCh_5Words_Input_Layout : STRUCT
        Signals_0 AT %B0 : WORD;
        Signals_1 AT %B2 : WORD;
        Signals_2 AT %B4 : WORD;
        Signals_3 AT %B6 : WORD;
        Signals_4 AT %B8 : WORD;
    END_STRUCT;
END_TYPE

TYPE
    rexroth_indradrive_ParamCh_5Words_Output_Layout : STRUCT
        Signals_5 AT %B0 : WORD;
        Signals_6 AT %B2 : WORD;
        Signals_7 AT %B4 : WORD;
        Signals_8 AT %B6 : WORD;
        Signals_9 AT %B8 : WORD;
    END_STRUCT;
END_TYPE

TYPE
    rexroth_press_Input_24_Words_Input_Layout : STRUCT
        Signals_0 AT %B0 : WORD;
        Signals_1 AT %B2 : WORD;
        Signals_2 AT %B4 : WORD;
        Signals_3 AT %B6 : WORD;
        Signals_4 AT %B8 : WORD;
        Signals_5 AT %B10 : WORD;
        Signals_6 AT %B12 : WORD;
        Signals_7 AT %B14 : WORD;
        Signals_8 AT %B16 : WORD;
        Signals_9 AT %B18 : WORD;
        Signals_10 AT %B20 : WORD;
        Signals_11 AT %B22 : WORD;
        Signals_12 AT %B24 : WORD;
        Signals_13 AT %B26 : WORD;
        Signals_14 AT %B28 : WORD;
        Signals_15 AT %B30 : WORD;
        Signals_16 AT %B32 : WORD;
        Signals_17 AT %B34 : WORD;
        Signals_18 AT %B36 : WORD;
        Signals_19 AT %B38 : WORD;
        Signals_20 AT %B40 : WORD;
        Signals_21 AT %B42 : WORD;
        Signals_22 AT %B44 : WORD;
        Signals_23 AT %B46 : WORD;
    END_STRUCT;
END_TYPE

TYPE
    rexroth_press_Output_21_Words_Output_Layout : STRUCT
        Signals_0 AT %B0 : WORD;
        Signals_1 AT %B2 : WORD;
        Signals_2 AT %B4 : WORD;
        Signals_3 AT %B6 : WORD;
        Signals_4 AT %B8 : WORD;
        Signals_5 AT %B10 : WORD;
        Signals_6 AT %B12 : WORD;
        Signals_7 AT %B14 : WORD;
        Signals_8 AT %B16 : WORD;
        Signals_9 AT %B18 : WORD;
        Signals_10 AT %B20 : WORD;
        Signals_11 AT %B22 : WORD;
        Signals_12 AT %B24 : WORD;
        Signals_13 AT %B26 : WORD;
        Signals_14 AT %B28 : WORD;
        Signals_15 AT %B30 : WORD;
        Signals_16 AT %B32 : WORD;
        Signals_17 AT %B34 : WORD;
        Signals_18 AT %B36 : WORD;
        Signals_19 AT %B38 : WORD;
        Signals_20 AT %B40 : WORD;
    END_STRUCT;
END_TYPE

TYPE
    rexroth_press_ParamCh_5Words_Input_Layout : STRUCT
        Signals_0 AT %B0 : WORD;
        Signals_1 AT %B2 : WORD;
        Signals_2 AT %B4 : WORD;
        Signals_3 AT %B6 : WORD;
        Signals_4 AT %B8 : WORD;
    END_STRUCT;
END_TYPE

TYPE
    rexroth_press_ParamCh_5Words_Output_Layout : STRUCT
        Signals_5 AT %B0 : WORD;
        Signals_6 AT %B2 : WORD;
        Signals_7 AT %B4 : WORD;
        Signals_8 AT %B6 : WORD;
        Signals_9 AT %B8 : WORD;
    END_STRUCT;
END_TYPE

TYPE
    rf186c_CM_1_Input_Layout : STRUCT
        Signals_0 AT %B0 : WORD;
    END_STRUCT;
END_TYPE

TYPE
    rf186c_CM_1_Output_Layout : STRUCT
        Signals_1 AT %B0 : WORD;
    END_STRUCT;
END_TYPE

TYPE
    rf186c_cyc_CM_Input_Layout : STRUCT
        Signals_0 AT %B0 : WORD;
    END_STRUCT;
END_TYPE

TYPE
    rf186c_cyc_CM_Output_Layout : STRUCT
        Signals_1 AT %B0 : WORD;
    END_STRUCT;
END_TYPE

TYPE
    rf186c_cyc_RF260R_1_Input_Layout : STRUCT
        Signals_0 AT %B0 : ARRAY[0..31] OF BYTE;
    END_STRUCT;
END_TYPE

TYPE
    rf186c_cyc_RF260R_1_Output_Layout : STRUCT
        Signals_1 AT %B0 : ARRAY[0..31] OF BYTE;
    END_STRUCT;
END_TYPE

TYPE
    rf186c_cyc_RF340R_1_Input_Layout : STRUCT
        Signals_0 AT %B0 : ARRAY[0..127] OF BYTE;
    END_STRUCT;
END_TYPE

TYPE
    rf186c_cyc_RF340R_1_Output_Layout : STRUCT
        Signals_1 AT %B0 : ARRAY[0..127] OF BYTE;
    END_STRUCT;
END_TYPE

TYPE
    rf186c_Reader_1_Input_Layout : STRUCT
        Signals_0 AT %B0 : WORD;
    END_STRUCT;
END_TYPE

TYPE
    rf186c_Reader_1_Output_Layout : STRUCT
        Signals_1 AT %B0 : WORD;
    END_STRUCT;
END_TYPE

TYPE
    smc_ex260_spn_16_Outputs16_Output_Layout : STRUCT
        Signals_0_0 AT %X0.0 : BOOL;
        Signals_0_1 AT %X0.1 : BOOL;
        Signals_0_2 AT %X0.2 : BOOL;
        Signals_0_3 AT %X0.3 : BOOL;
        Signals_0_4 AT %X0.4 : BOOL;
        Signals_0_5 AT %X0.5 : BOOL;
        Signals_0_6 AT %X0.6 : BOOL;
        Signals_0_7 AT %X0.7 : BOOL;
        Signals_1_0 AT %X1.0 : BOOL;
        Signals_1_1 AT %X1.1 : BOOL;
        Signals_1_2 AT %X1.2 : BOOL;
        Signals_1_3 AT %X1.3 : BOOL;
        Signals_1_4 AT %X1.4 : BOOL;
        Signals_1_5 AT %X1.5 : BOOL;
        Signals_1_6 AT %X1.6 : BOOL;
        Signals_1_7 AT %X1.7 : BOOL;
    END_STRUCT;
END_TYPE

TYPE
    smc_ex260_spn_32_Outputs32_Output_Layout : STRUCT
        Signals_0_0 AT %X0.0 : BOOL;
        Signals_0_1 AT %X0.1 : BOOL;
        Signals_0_2 AT %X0.2 : BOOL;
        Signals_0_3 AT %X0.3 : BOOL;
        Signals_0_4 AT %X0.4 : BOOL;
        Signals_0_5 AT %X0.5 : BOOL;
        Signals_0_6 AT %X0.6 : BOOL;
        Signals_0_7 AT %X0.7 : BOOL;
        Signals_1_0 AT %X1.0 : BOOL;
        Signals_1_1 AT %X1.1 : BOOL;
        Signals_1_2 AT %X1.2 : BOOL;
        Signals_1_3 AT %X1.3 : BOOL;
        Signals_1_4 AT %X1.4 : BOOL;
        Signals_1_5 AT %X1.5 : BOOL;
        Signals_1_6 AT %X1.6 : BOOL;
        Signals_1_7 AT %X1.7 : BOOL;
        Signals_2_0 AT %X2.0 : BOOL;
        Signals_2_1 AT %X2.1 : BOOL;
        Signals_2_2 AT %X2.2 : BOOL;
        Signals_2_3 AT %X2.3 : BOOL;
        Signals_2_4 AT %X2.4 : BOOL;
        Signals_2_5 AT %X2.5 : BOOL;
        Signals_2_6 AT %X2.6 : BOOL;
        Signals_2_7 AT %X2.7 : BOOL;
        Signals_3_0 AT %X3.0 : BOOL;
        Signals_3_1 AT %X3.1 : BOOL;
        Signals_3_2 AT %X3.2 : BOOL;
        Signals_3_3 AT %X3.3 : BOOL;
        Signals_3_4 AT %X3.4 : BOOL;
        Signals_3_5 AT %X3.5 : BOOL;
        Signals_3_6 AT %X3.6 : BOOL;
        Signals_3_7 AT %X3.7 : BOOL;
    END_STRUCT;
END_TYPE

TYPE
    ureol2l_1_T2O_State_Input_Layout : STRUCT
        Signals_0_0 AT %X0.0 : BOOL;
        Signals_0_1 AT %X0.1 : BOOL;
        Signals_0_2 AT %X0.2 : BOOL;
        Signals_0_3 AT %X0.3 : BOOL;
        Signals_0_4 AT %X0.4 : BOOL;
        Signals_0_5 AT %X0.5 : BOOL;
        Signals_0_6 AT %X0.6 : BOOL;
        Signals_0_7 AT %X0.7 : BOOL;
        Signals_0_8 AT %X1.0 : BOOL;
        Signals_0_9 AT %X1.1 : BOOL;
        Signals_0_10 AT %X1.2 : BOOL;
        Signals_0_11 AT %X1.3 : BOOL;
        Signals_0_12 AT %X1.4 : BOOL;
        Signals_0_13 AT %X1.5 : BOOL;
        Signals_0_14 AT %X1.6 : BOOL;
        Signals_0_15 AT %X1.7 : BOOL;
        Signals_0_16 AT %X2.0 : BOOL;
        Signals_0_17 AT %X2.1 : BOOL;
        Signals_0_18 AT %X2.2 : BOOL;
        Signals_0_19 AT %X2.3 : BOOL;
        Signals_0_20 AT %X2.4 : BOOL;
        Signals_0_21 AT %X2.5 : BOOL;
        Signals_0_22 AT %X2.6 : BOOL;
        Signals_0_23 AT %X2.7 : BOOL;
        Signals_0_24 AT %X3.0 : BOOL;
        Signals_0_25 AT %X3.1 : BOOL;
        Signals_0_26 AT %X3.2 : BOOL;
        Signals_0_27 AT %X3.3 : BOOL;
        Signals_0_28 AT %X3.4 : BOOL;
        Signals_0_29 AT %X3.5 : BOOL;
        Signals_0_30 AT %X3.6 : BOOL;
        Signals_0_31 AT %X3.7 : BOOL;
        Signals_0_32 AT %X4.0 : BOOL;
        Signals_0_33 AT %X4.1 : BOOL;
        Signals_0_34 AT %X4.2 : BOOL;
        Signals_0_35 AT %X4.3 : BOOL;
        Signals_0_36 AT %X4.4 : BOOL;
        Signals_0_37 AT %X4.5 : BOOL;
        Signals_0_38 AT %X4.6 : BOOL;
        Signals_0_39 AT %X4.7 : BOOL;
        Signals_0_40 AT %X5.0 : BOOL;
        Signals_0_41 AT %X5.1 : BOOL;
        Signals_0_42 AT %X5.2 : BOOL;
        Signals_0_43 AT %X5.3 : BOOL;
        Signals_0_44 AT %X5.4 : BOOL;
        Signals_0_45 AT %X5.5 : BOOL;
        Signals_0_46 AT %X5.6 : BOOL;
        Signals_0_47 AT %X5.7 : BOOL;
        Signals_0_48 AT %X6.0 : BOOL;
        Signals_0_49 AT %X6.1 : BOOL;
        Signals_0_50 AT %X6.2 : BOOL;
        Signals_0_51 AT %X6.3 : BOOL;
        Signals_0_52 AT %X6.4 : BOOL;
        Signals_0_53 AT %X6.5 : BOOL;
        Signals_0_54 AT %X6.6 : BOOL;
        Signals_0_55 AT %X6.7 : BOOL;
        Signals_0_56 AT %X7.0 : BOOL;
        Signals_0_57 AT %X7.1 : BOOL;
        Signals_0_58 AT %X7.2 : BOOL;
        Signals_0_59 AT %X7.3 : BOOL;
        Signals_0_60 AT %X7.4 : BOOL;
        Signals_0_61 AT %X7.5 : BOOL;
        Signals_0_62 AT %X7.6 : BOOL;
        Signals_0_63 AT %X7.7 : BOOL;
        Signals_0_64 AT %X8.0 : BOOL;
        Signals_0_65 AT %X8.1 : BOOL;
        Signals_0_66 AT %X8.2 : BOOL;
        Signals_0_67 AT %X8.3 : BOOL;
        Signals_0_68 AT %X8.4 : BOOL;
        Signals_0_69 AT %X8.5 : BOOL;
        Signals_0_70 AT %X8.6 : BOOL;
        Signals_0_71 AT %X8.7 : BOOL;
        Signals_0_72 AT %X9.0 : BOOL;
        Signals_0_73 AT %X9.1 : BOOL;
        Signals_0_74 AT %X9.2 : BOOL;
        Signals_0_75 AT %X9.3 : BOOL;
        Signals_0_76 AT %X9.4 : BOOL;
        Signals_0_77 AT %X9.5 : BOOL;
        Signals_0_78 AT %X9.6 : BOOL;
        Signals_0_79 AT %X9.7 : BOOL;
        Signals_0_80 AT %X10.0 : BOOL;
        Signals_0_81 AT %X10.1 : BOOL;
        Signals_0_82 AT %X10.2 : BOOL;
        Signals_0_83 AT %X10.3 : BOOL;
        Signals_0_84 AT %X10.4 : BOOL;
        Signals_0_85 AT %X10.5 : BOOL;
        Signals_0_86 AT %X10.6 : BOOL;
        Signals_0_87 AT %X10.7 : BOOL;
        Signals_0_88 AT %X11.0 : BOOL;
        Signals_0_89 AT %X11.1 : BOOL;
        Signals_0_90 AT %X11.2 : BOOL;
        Signals_0_91 AT %X11.3 : BOOL;
        Signals_0_92 AT %X11.4 : BOOL;
        Signals_0_93 AT %X11.5 : BOOL;
        Signals_0_94 AT %X11.6 : BOOL;
        Signals_0_95 AT %X11.7 : BOOL;
        Signals_0_96 AT %X12.0 : BOOL;
        Signals_0_97 AT %X12.1 : BOOL;
        Signals_0_98 AT %X12.2 : BOOL;
        Signals_0_99 AT %X12.3 : BOOL;
        Signals_0_100 AT %X12.4 : BOOL;
        Signals_0_101 AT %X12.5 : BOOL;
        Signals_0_102 AT %X12.6 : BOOL;
        Signals_0_103 AT %X12.7 : BOOL;
        Signals_0_104 AT %X13.0 : BOOL;
        Signals_0_105 AT %X13.1 : BOOL;
        Signals_0_106 AT %X13.2 : BOOL;
        Signals_0_107 AT %X13.3 : BOOL;
        Signals_0_108 AT %X13.4 : BOOL;
        Signals_0_109 AT %X13.5 : BOOL;
        Signals_0_110 AT %X13.6 : BOOL;
        Signals_0_111 AT %X13.7 : BOOL;
        Signals_0_112 AT %X14.0 : BOOL;
        Signals_0_113 AT %X14.1 : BOOL;
        Signals_0_114 AT %X14.2 : BOOL;
        Signals_0_115 AT %X14.3 : BOOL;
        Signals_0_116 AT %X14.4 : BOOL;
        Signals_0_117 AT %X14.5 : BOOL;
        Signals_0_118 AT %X14.6 : BOOL;
        Signals_0_119 AT %X14.7 : BOOL;
        Signals_0_120 AT %X15.0 : BOOL;
        Signals_0_121 AT %X15.1 : BOOL;
        Signals_0_122 AT %X15.2 : BOOL;
        Signals_0_123 AT %X15.3 : BOOL;
        Signals_0_124 AT %X15.4 : BOOL;
        Signals_0_125 AT %X15.5 : BOOL;
        Signals_0_126 AT %X15.6 : BOOL;
        Signals_0_127 AT %X15.7 : BOOL;
        Signals_0_128 AT %X16.0 : BOOL;
        Signals_0_129 AT %X16.1 : BOOL;
        Signals_0_130 AT %X16.2 : BOOL;
        Signals_0_131 AT %X16.3 : BOOL;
        Signals_0_132 AT %X16.4 : BOOL;
        Signals_0_133 AT %X16.5 : BOOL;
        Signals_0_134 AT %X16.6 : BOOL;
        Signals_0_135 AT %X16.7 : BOOL;
        Signals_0_136 AT %X17.0 : BOOL;
        Signals_0_137 AT %X17.1 : BOOL;
        Signals_0_138 AT %X17.2 : BOOL;
        Signals_0_139 AT %X17.3 : BOOL;
        Signals_0_140 AT %X17.4 : BOOL;
        Signals_0_141 AT %X17.5 : BOOL;
        Signals_0_142 AT %X17.6 : BOOL;
        Signals_0_143 AT %X17.7 : BOOL;
        Signals_0_144 AT %X18.0 : BOOL;
        Signals_0_145 AT %X18.1 : BOOL;
        Signals_0_146 AT %X18.2 : BOOL;
        Signals_0_147 AT %X18.3 : BOOL;
        Signals_0_148 AT %X18.4 : BOOL;
        Signals_0_149 AT %X18.5 : BOOL;
        Signals_0_150 AT %X18.6 : BOOL;
        Signals_0_151 AT %X18.7 : BOOL;
        Signals_0_152 AT %X19.0 : BOOL;
        Signals_0_153 AT %X19.1 : BOOL;
        Signals_0_154 AT %X19.2 : BOOL;
        Signals_0_155 AT %X19.3 : BOOL;
        Signals_0_156 AT %X19.4 : BOOL;
        Signals_0_157 AT %X19.5 : BOOL;
        Signals_0_158 AT %X19.6 : BOOL;
        Signals_0_159 AT %X19.7 : BOOL;
        Signals_0_160 AT %X20.0 : BOOL;
        Signals_0_161 AT %X20.1 : BOOL;
        Signals_0_162 AT %X20.2 : BOOL;
        Signals_0_163 AT %X20.3 : BOOL;
        Signals_0_164 AT %X20.4 : BOOL;
        Signals_0_165 AT %X20.5 : BOOL;
        Signals_0_166 AT %X20.6 : BOOL;
        Signals_0_167 AT %X20.7 : BOOL;
        Signals_0_168 AT %X21.0 : BOOL;
        Signals_0_169 AT %X21.1 : BOOL;
        Signals_0_170 AT %X21.2 : BOOL;
        Signals_0_171 AT %X21.3 : BOOL;
        Signals_0_172 AT %X21.4 : BOOL;
        Signals_0_173 AT %X21.5 : BOOL;
        Signals_0_174 AT %X21.6 : BOOL;
        Signals_0_175 AT %X21.7 : BOOL;
        Signals_0_176 AT %X22.0 : BOOL;
        Signals_0_177 AT %X22.1 : BOOL;
        Signals_0_178 AT %X22.2 : BOOL;
        Signals_0_179 AT %X22.3 : BOOL;
        Signals_0_180 AT %X22.4 : BOOL;
        Signals_0_181 AT %X22.5 : BOOL;
        Signals_0_182 AT %X22.6 : BOOL;
        Signals_0_183 AT %X22.7 : BOOL;
        Signals_0_184 AT %X23.0 : BOOL;
        Signals_0_185 AT %X23.1 : BOOL;
        Signals_0_186 AT %X23.2 : BOOL;
        Signals_0_187 AT %X23.3 : BOOL;
        Signals_0_188 AT %X23.4 : BOOL;
        Signals_0_189 AT %X23.5 : BOOL;
        Signals_0_190 AT %X23.6 : BOOL;
        Signals_0_191 AT %X23.7 : BOOL;
        Signals_0_192 AT %X24.0 : BOOL;
        Signals_0_193 AT %X24.1 : BOOL;
        Signals_0_194 AT %X24.2 : BOOL;
        Signals_0_195 AT %X24.3 : BOOL;
        Signals_0_196 AT %X24.4 : BOOL;
        Signals_0_197 AT %X24.5 : BOOL;
        Signals_0_198 AT %X24.6 : BOOL;
        Signals_0_199 AT %X24.7 : BOOL;
        Signals_0_200 AT %X25.0 : BOOL;
        Signals_0_201 AT %X25.1 : BOOL;
        Signals_0_202 AT %X25.2 : BOOL;
        Signals_0_203 AT %X25.3 : BOOL;
        Signals_0_204 AT %X25.4 : BOOL;
        Signals_0_205 AT %X25.5 : BOOL;
        Signals_0_206 AT %X25.6 : BOOL;
        Signals_0_207 AT %X25.7 : BOOL;
        Signals_0_208 AT %X26.0 : BOOL;
        Signals_0_209 AT %X26.1 : BOOL;
        Signals_0_210 AT %X26.2 : BOOL;
        Signals_0_211 AT %X26.3 : BOOL;
        Signals_0_212 AT %X26.4 : BOOL;
        Signals_0_213 AT %X26.5 : BOOL;
        Signals_0_214 AT %X26.6 : BOOL;
        Signals_0_215 AT %X26.7 : BOOL;
        Signals_0_216 AT %X27.0 : BOOL;
        Signals_0_217 AT %X27.1 : BOOL;
        Signals_0_218 AT %X27.2 : BOOL;
        Signals_0_219 AT %X27.3 : BOOL;
        Signals_0_220 AT %X27.4 : BOOL;
        Signals_0_221 AT %X27.5 : BOOL;
        Signals_0_222 AT %X27.6 : BOOL;
        Signals_0_223 AT %X27.7 : BOOL;
        Signals_0_224 AT %X28.0 : BOOL;
        Signals_0_225 AT %X28.1 : BOOL;
        Signals_0_226 AT %X28.2 : BOOL;
        Signals_0_227 AT %X28.3 : BOOL;
        Signals_0_228 AT %X28.4 : BOOL;
        Signals_0_229 AT %X28.5 : BOOL;
        Signals_0_230 AT %X28.6 : BOOL;
        Signals_0_231 AT %X28.7 : BOOL;
        Signals_0_232 AT %X29.0 : BOOL;
        Signals_0_233 AT %X29.1 : BOOL;
        Signals_0_234 AT %X29.2 : BOOL;
        Signals_0_235 AT %X29.3 : BOOL;
        Signals_0_236 AT %X29.4 : BOOL;
        Signals_0_237 AT %X29.5 : BOOL;
        Signals_0_238 AT %X29.6 : BOOL;
        Signals_0_239 AT %X29.7 : BOOL;
        Signals_0_240 AT %X30.0 : BOOL;
        Signals_0_241 AT %X30.1 : BOOL;
        Signals_0_242 AT %X30.2 : BOOL;
        Signals_0_243 AT %X30.3 : BOOL;
        Signals_0_244 AT %X30.4 : BOOL;
        Signals_0_245 AT %X30.5 : BOOL;
        Signals_0_246 AT %X30.6 : BOOL;
        Signals_0_247 AT %X30.7 : BOOL;
        Signals_0_248 AT %X31.0 : BOOL;
        Signals_0_249 AT %X31.1 : BOOL;
        Signals_0_250 AT %X31.2 : BOOL;
        Signals_0_251 AT %X31.3 : BOOL;
        Signals_0_252 AT %X31.4 : BOOL;
        Signals_0_253 AT %X31.5 : BOOL;
        Signals_0_254 AT %X31.6 : BOOL;
        Signals_0_255 AT %X31.7 : BOOL;
    END_STRUCT;
END_TYPE

TYPE
    ureol2l_10_O2T_General_Purpose_Registers_2_Output_Layout : STRUCT
        Signals_0 AT %B0 : ARRAY[0..799] OF BOOL;
    END_STRUCT;
END_TYPE

TYPE
    ureol2l_2_T2O_IO_Input_Layout : STRUCT
        Signals_0 AT %B0 : ARRAY[0..543] OF BOOL;
    END_STRUCT;
END_TYPE

TYPE
    ureol2l_3_T2O_Joints_Input_Layout : STRUCT
        Signals_0 AT %B0 : ARRAY[0..831] OF BOOL;
    END_STRUCT;
END_TYPE

TYPE
    ureol2l_4_T2O_TCP_Input_Layout : STRUCT
        Signals_0 AT %B0 : ARRAY[0..607] OF BOOL;
    END_STRUCT;
END_TYPE

TYPE
    ureol2l_5_T2O_General_Purpose_Bit_Registers_Input_Layout : STRUCT
        Signals_0_0 AT %X0.0 : BOOL;
        Signals_0_1 AT %X0.1 : BOOL;
        Signals_0_2 AT %X0.2 : BOOL;
        Signals_0_3 AT %X0.3 : BOOL;
        Signals_0_4 AT %X0.4 : BOOL;
        Signals_0_5 AT %X0.5 : BOOL;
        Signals_0_6 AT %X0.6 : BOOL;
        Signals_0_7 AT %X0.7 : BOOL;
        Signals_0_8 AT %X1.0 : BOOL;
        Signals_0_9 AT %X1.1 : BOOL;
        Signals_0_10 AT %X1.2 : BOOL;
        Signals_0_11 AT %X1.3 : BOOL;
        Signals_0_12 AT %X1.4 : BOOL;
        Signals_0_13 AT %X1.5 : BOOL;
        Signals_0_14 AT %X1.6 : BOOL;
        Signals_0_15 AT %X1.7 : BOOL;
        Signals_0_16 AT %X2.0 : BOOL;
        Signals_0_17 AT %X2.1 : BOOL;
        Signals_0_18 AT %X2.2 : BOOL;
        Signals_0_19 AT %X2.3 : BOOL;
        Signals_0_20 AT %X2.4 : BOOL;
        Signals_0_21 AT %X2.5 : BOOL;
        Signals_0_22 AT %X2.6 : BOOL;
        Signals_0_23 AT %X2.7 : BOOL;
        Signals_0_24 AT %X3.0 : BOOL;
        Signals_0_25 AT %X3.1 : BOOL;
        Signals_0_26 AT %X3.2 : BOOL;
        Signals_0_27 AT %X3.3 : BOOL;
        Signals_0_28 AT %X3.4 : BOOL;
        Signals_0_29 AT %X3.5 : BOOL;
        Signals_0_30 AT %X3.6 : BOOL;
        Signals_0_31 AT %X3.7 : BOOL;
        Signals_0_32 AT %X4.0 : BOOL;
        Signals_0_33 AT %X4.1 : BOOL;
        Signals_0_34 AT %X4.2 : BOOL;
        Signals_0_35 AT %X4.3 : BOOL;
        Signals_0_36 AT %X4.4 : BOOL;
        Signals_0_37 AT %X4.5 : BOOL;
        Signals_0_38 AT %X4.6 : BOOL;
        Signals_0_39 AT %X4.7 : BOOL;
        Signals_0_40 AT %X5.0 : BOOL;
        Signals_0_41 AT %X5.1 : BOOL;
        Signals_0_42 AT %X5.2 : BOOL;
        Signals_0_43 AT %X5.3 : BOOL;
        Signals_0_44 AT %X5.4 : BOOL;
        Signals_0_45 AT %X5.5 : BOOL;
        Signals_0_46 AT %X5.6 : BOOL;
        Signals_0_47 AT %X5.7 : BOOL;
        Signals_0_48 AT %X6.0 : BOOL;
        Signals_0_49 AT %X6.1 : BOOL;
        Signals_0_50 AT %X6.2 : BOOL;
        Signals_0_51 AT %X6.3 : BOOL;
        Signals_0_52 AT %X6.4 : BOOL;
        Signals_0_53 AT %X6.5 : BOOL;
        Signals_0_54 AT %X6.6 : BOOL;
        Signals_0_55 AT %X6.7 : BOOL;
        Signals_0_56 AT %X7.0 : BOOL;
        Signals_0_57 AT %X7.1 : BOOL;
        Signals_0_58 AT %X7.2 : BOOL;
        Signals_0_59 AT %X7.3 : BOOL;
        Signals_0_60 AT %X7.4 : BOOL;
        Signals_0_61 AT %X7.5 : BOOL;
        Signals_0_62 AT %X7.6 : BOOL;
        Signals_0_63 AT %X7.7 : BOOL;
    END_STRUCT;
END_TYPE

TYPE
    ureol2l_6_T2O_General_Purpose_Int_Registers_Input_Layout : STRUCT
        Signals_0 AT %B0 : ARRAY[0..767] OF BOOL;
    END_STRUCT;
END_TYPE

TYPE
    ureol2l_7_T2O_General_Purpose_Float_Registers_Input_Layout : STRUCT
        Signals_0 AT %B0 : ARRAY[0..767] OF BOOL;
    END_STRUCT;
END_TYPE

TYPE
    ureol2l_8_O2T_Robot_IO_Output_Layout : STRUCT
        Signals_0_0 AT %X0.0 : BOOL;
        Signals_0_1 AT %X0.1 : BOOL;
        Signals_0_2 AT %X0.2 : BOOL;
        Signals_0_3 AT %X0.3 : BOOL;
        Signals_0_4 AT %X0.4 : BOOL;
        Signals_0_5 AT %X0.5 : BOOL;
        Signals_0_6 AT %X0.6 : BOOL;
        Signals_0_7 AT %X0.7 : BOOL;
        Signals_0_8 AT %X1.0 : BOOL;
        Signals_0_9 AT %X1.1 : BOOL;
        Signals_0_10 AT %X1.2 : BOOL;
        Signals_0_11 AT %X1.3 : BOOL;
        Signals_0_12 AT %X1.4 : BOOL;
        Signals_0_13 AT %X1.5 : BOOL;
        Signals_0_14 AT %X1.6 : BOOL;
        Signals_0_15 AT %X1.7 : BOOL;
        Signals_0_16 AT %X2.0 : BOOL;
        Signals_0_17 AT %X2.1 : BOOL;
        Signals_0_18 AT %X2.2 : BOOL;
        Signals_0_19 AT %X2.3 : BOOL;
        Signals_0_20 AT %X2.4 : BOOL;
        Signals_0_21 AT %X2.5 : BOOL;
        Signals_0_22 AT %X2.6 : BOOL;
        Signals_0_23 AT %X2.7 : BOOL;
        Signals_0_24 AT %X3.0 : BOOL;
        Signals_0_25 AT %X3.1 : BOOL;
        Signals_0_26 AT %X3.2 : BOOL;
        Signals_0_27 AT %X3.3 : BOOL;
        Signals_0_28 AT %X3.4 : BOOL;
        Signals_0_29 AT %X3.5 : BOOL;
        Signals_0_30 AT %X3.6 : BOOL;
        Signals_0_31 AT %X3.7 : BOOL;
        Signals_0_32 AT %X4.0 : BOOL;
        Signals_0_33 AT %X4.1 : BOOL;
        Signals_0_34 AT %X4.2 : BOOL;
        Signals_0_35 AT %X4.3 : BOOL;
        Signals_0_36 AT %X4.4 : BOOL;
        Signals_0_37 AT %X4.5 : BOOL;
        Signals_0_38 AT %X4.6 : BOOL;
        Signals_0_39 AT %X4.7 : BOOL;
        Signals_0_40 AT %X5.0 : BOOL;
        Signals_0_41 AT %X5.1 : BOOL;
        Signals_0_42 AT %X5.2 : BOOL;
        Signals_0_43 AT %X5.3 : BOOL;
        Signals_0_44 AT %X5.4 : BOOL;
        Signals_0_45 AT %X5.5 : BOOL;
        Signals_0_46 AT %X5.6 : BOOL;
        Signals_0_47 AT %X5.7 : BOOL;
        Signals_0_48 AT %X6.0 : BOOL;
        Signals_0_49 AT %X6.1 : BOOL;
        Signals_0_50 AT %X6.2 : BOOL;
        Signals_0_51 AT %X6.3 : BOOL;
        Signals_0_52 AT %X6.4 : BOOL;
        Signals_0_53 AT %X6.5 : BOOL;
        Signals_0_54 AT %X6.6 : BOOL;
        Signals_0_55 AT %X6.7 : BOOL;
        Signals_0_56 AT %X7.0 : BOOL;
        Signals_0_57 AT %X7.1 : BOOL;
        Signals_0_58 AT %X7.2 : BOOL;
        Signals_0_59 AT %X7.3 : BOOL;
        Signals_0_60 AT %X7.4 : BOOL;
        Signals_0_61 AT %X7.5 : BOOL;
        Signals_0_62 AT %X7.6 : BOOL;
        Signals_0_63 AT %X7.7 : BOOL;
        Signals_0_64 AT %X8.0 : BOOL;
        Signals_0_65 AT %X8.1 : BOOL;
        Signals_0_66 AT %X8.2 : BOOL;
        Signals_0_67 AT %X8.3 : BOOL;
        Signals_0_68 AT %X8.4 : BOOL;
        Signals_0_69 AT %X8.5 : BOOL;
        Signals_0_70 AT %X8.6 : BOOL;
        Signals_0_71 AT %X8.7 : BOOL;
        Signals_0_72 AT %X9.0 : BOOL;
        Signals_0_73 AT %X9.1 : BOOL;
        Signals_0_74 AT %X9.2 : BOOL;
        Signals_0_75 AT %X9.3 : BOOL;
        Signals_0_76 AT %X9.4 : BOOL;
        Signals_0_77 AT %X9.5 : BOOL;
        Signals_0_78 AT %X9.6 : BOOL;
        Signals_0_79 AT %X9.7 : BOOL;
        Signals_0_80 AT %X10.0 : BOOL;
        Signals_0_81 AT %X10.1 : BOOL;
        Signals_0_82 AT %X10.2 : BOOL;
        Signals_0_83 AT %X10.3 : BOOL;
        Signals_0_84 AT %X10.4 : BOOL;
        Signals_0_85 AT %X10.5 : BOOL;
        Signals_0_86 AT %X10.6 : BOOL;
        Signals_0_87 AT %X10.7 : BOOL;
        Signals_0_88 AT %X11.0 : BOOL;
        Signals_0_89 AT %X11.1 : BOOL;
        Signals_0_90 AT %X11.2 : BOOL;
        Signals_0_91 AT %X11.3 : BOOL;
        Signals_0_92 AT %X11.4 : BOOL;
        Signals_0_93 AT %X11.5 : BOOL;
        Signals_0_94 AT %X11.6 : BOOL;
        Signals_0_95 AT %X11.7 : BOOL;
        Signals_0_96 AT %X12.0 : BOOL;
        Signals_0_97 AT %X12.1 : BOOL;
        Signals_0_98 AT %X12.2 : BOOL;
        Signals_0_99 AT %X12.3 : BOOL;
        Signals_0_100 AT %X12.4 : BOOL;
        Signals_0_101 AT %X12.5 : BOOL;
        Signals_0_102 AT %X12.6 : BOOL;
        Signals_0_103 AT %X12.7 : BOOL;
        Signals_0_104 AT %X13.0 : BOOL;
        Signals_0_105 AT %X13.1 : BOOL;
        Signals_0_106 AT %X13.2 : BOOL;
        Signals_0_107 AT %X13.3 : BOOL;
        Signals_0_108 AT %X13.4 : BOOL;
        Signals_0_109 AT %X13.5 : BOOL;
        Signals_0_110 AT %X13.6 : BOOL;
        Signals_0_111 AT %X13.7 : BOOL;
        Signals_0_112 AT %X14.0 : BOOL;
        Signals_0_113 AT %X14.1 : BOOL;
        Signals_0_114 AT %X14.2 : BOOL;
        Signals_0_115 AT %X14.3 : BOOL;
        Signals_0_116 AT %X14.4 : BOOL;
        Signals_0_117 AT %X14.5 : BOOL;
        Signals_0_118 AT %X14.6 : BOOL;
        Signals_0_119 AT %X14.7 : BOOL;
        Signals_0_120 AT %X15.0 : BOOL;
        Signals_0_121 AT %X15.1 : BOOL;
        Signals_0_122 AT %X15.2 : BOOL;
        Signals_0_123 AT %X15.3 : BOOL;
        Signals_0_124 AT %X15.4 : BOOL;
        Signals_0_125 AT %X15.5 : BOOL;
        Signals_0_126 AT %X15.6 : BOOL;
        Signals_0_127 AT %X15.7 : BOOL;
        Signals_0_128 AT %X16.0 : BOOL;
        Signals_0_129 AT %X16.1 : BOOL;
        Signals_0_130 AT %X16.2 : BOOL;
        Signals_0_131 AT %X16.3 : BOOL;
        Signals_0_132 AT %X16.4 : BOOL;
        Signals_0_133 AT %X16.5 : BOOL;
        Signals_0_134 AT %X16.6 : BOOL;
        Signals_0_135 AT %X16.7 : BOOL;
        Signals_0_136 AT %X17.0 : BOOL;
        Signals_0_137 AT %X17.1 : BOOL;
        Signals_0_138 AT %X17.2 : BOOL;
        Signals_0_139 AT %X17.3 : BOOL;
        Signals_0_140 AT %X17.4 : BOOL;
        Signals_0_141 AT %X17.5 : BOOL;
        Signals_0_142 AT %X17.6 : BOOL;
        Signals_0_143 AT %X17.7 : BOOL;
        Signals_0_144 AT %X18.0 : BOOL;
        Signals_0_145 AT %X18.1 : BOOL;
        Signals_0_146 AT %X18.2 : BOOL;
        Signals_0_147 AT %X18.3 : BOOL;
        Signals_0_148 AT %X18.4 : BOOL;
        Signals_0_149 AT %X18.5 : BOOL;
        Signals_0_150 AT %X18.6 : BOOL;
        Signals_0_151 AT %X18.7 : BOOL;
        Signals_0_152 AT %X19.0 : BOOL;
        Signals_0_153 AT %X19.1 : BOOL;
        Signals_0_154 AT %X19.2 : BOOL;
        Signals_0_155 AT %X19.3 : BOOL;
        Signals_0_156 AT %X19.4 : BOOL;
        Signals_0_157 AT %X19.5 : BOOL;
        Signals_0_158 AT %X19.6 : BOOL;
        Signals_0_159 AT %X19.7 : BOOL;
        Signals_0_160 AT %X20.0 : BOOL;
        Signals_0_161 AT %X20.1 : BOOL;
        Signals_0_162 AT %X20.2 : BOOL;
        Signals_0_163 AT %X20.3 : BOOL;
        Signals_0_164 AT %X20.4 : BOOL;
        Signals_0_165 AT %X20.5 : BOOL;
        Signals_0_166 AT %X20.6 : BOOL;
        Signals_0_167 AT %X20.7 : BOOL;
        Signals_0_168 AT %X21.0 : BOOL;
        Signals_0_169 AT %X21.1 : BOOL;
        Signals_0_170 AT %X21.2 : BOOL;
        Signals_0_171 AT %X21.3 : BOOL;
        Signals_0_172 AT %X21.4 : BOOL;
        Signals_0_173 AT %X21.5 : BOOL;
        Signals_0_174 AT %X21.6 : BOOL;
        Signals_0_175 AT %X21.7 : BOOL;
        Signals_0_176 AT %X22.0 : BOOL;
        Signals_0_177 AT %X22.1 : BOOL;
        Signals_0_178 AT %X22.2 : BOOL;
        Signals_0_179 AT %X22.3 : BOOL;
        Signals_0_180 AT %X22.4 : BOOL;
        Signals_0_181 AT %X22.5 : BOOL;
        Signals_0_182 AT %X22.6 : BOOL;
        Signals_0_183 AT %X22.7 : BOOL;
        Signals_0_184 AT %X23.0 : BOOL;
        Signals_0_185 AT %X23.1 : BOOL;
        Signals_0_186 AT %X23.2 : BOOL;
        Signals_0_187 AT %X23.3 : BOOL;
        Signals_0_188 AT %X23.4 : BOOL;
        Signals_0_189 AT %X23.5 : BOOL;
        Signals_0_190 AT %X23.6 : BOOL;
        Signals_0_191 AT %X23.7 : BOOL;
    END_STRUCT;
END_TYPE
